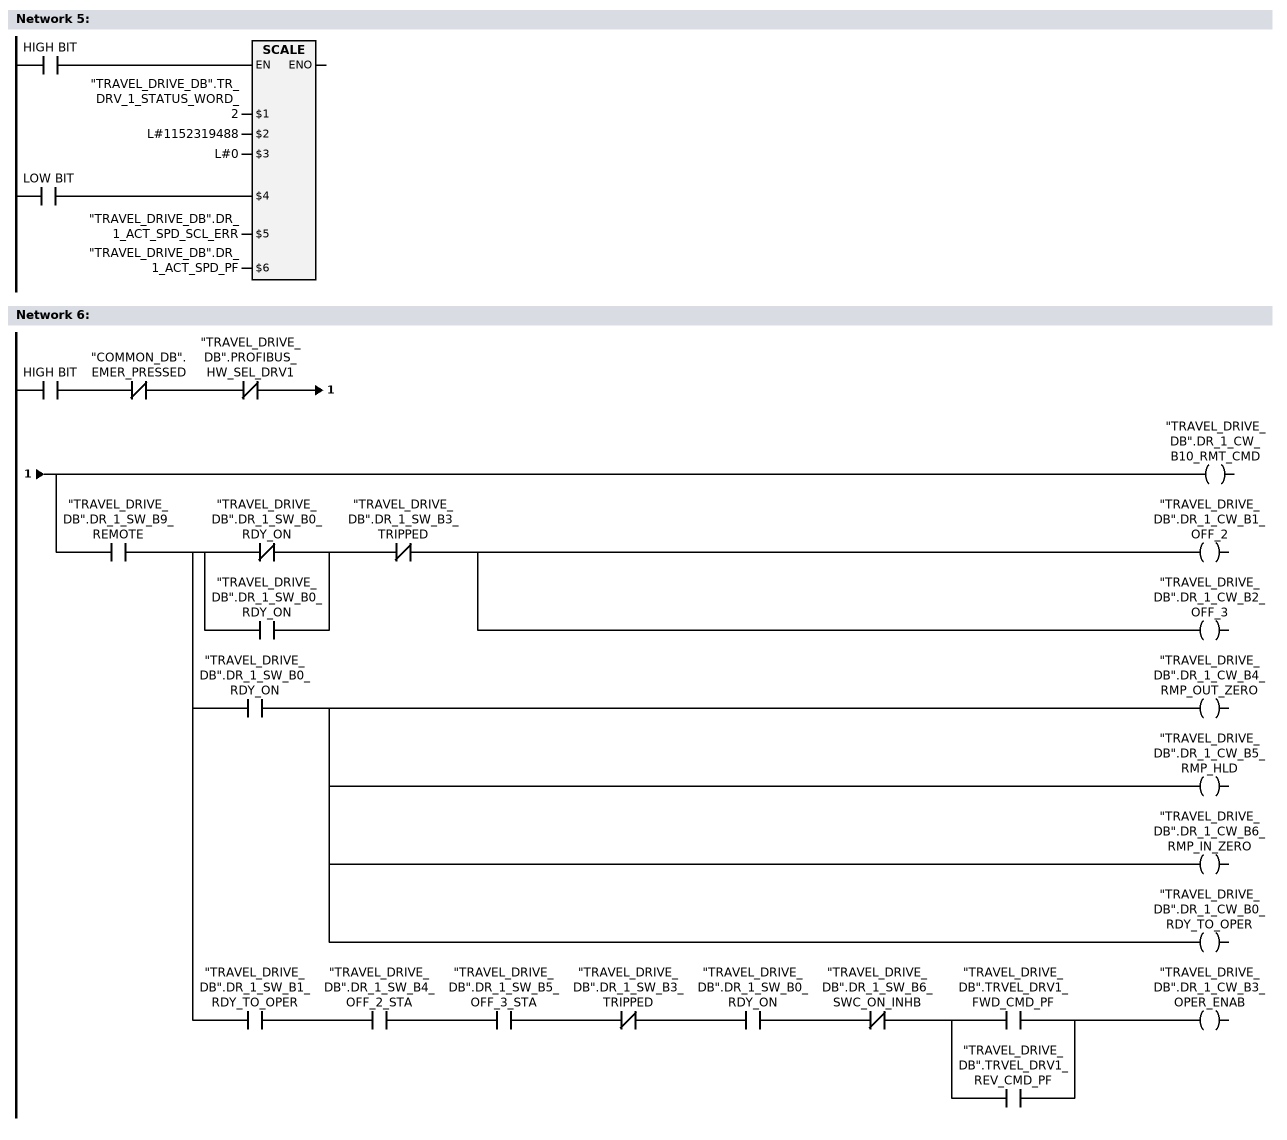
NETWORK
TITLE =
      A     "LOW BIT";
      =     L 22.0;
      BLD   103;
      A     "HIGH BIT";
      JNB   M007;
      CALL  "SCALE" (
           $1                       := "TRAVEL_DRIVE_DB".TR_DRV_1_STATUS_WORD_2,
           $2                       := L#1152319488,
           $3                       := L#0,
           $4                       := L 22.0,
           $5                       := "TRAVEL_DRIVE_DB".DR_1_ACT_SPD_SCL_ERR,
           $6                       := "TRAVEL_DRIVE_DB".DR_1_ACT_SPD_PF);
M007: NOP   0;
NETWORK
TITLE =
      A     "HIGH BIT";
      AN    "COMMON_DB".EMER_PRESSED;
      AN    "TRAVEL_DRIVE_DB".PROFIBUS_HW_SEL_DRV1;
      =     L 22.0;
      A     L 22.0;
      BLD   102;
      =     "TRAVEL_DRIVE_DB".DR_1_CW_B10_RMT_CMD;
      A     L 22.0;
      A     "TRAVEL_DRIVE_DB".DR_1_SW_B9_REMOTE;
      =     L 22.1;
      A     L 22.1;
      A(;
      ON    "TRAVEL_DRIVE_DB".DR_1_SW_B0_RDY_ON;
      O     "TRAVEL_DRIVE_DB".DR_1_SW_B0_RDY_ON;
      );
      AN    "TRAVEL_DRIVE_DB".DR_1_SW_B3_TRIPPED;
      =     "TRAVEL_DRIVE_DB".DR_1_CW_B1_OFF_2;
      =     "TRAVEL_DRIVE_DB".DR_1_CW_B2_OFF_3;
      A     L 22.1;
      A     "TRAVEL_DRIVE_DB".DR_1_SW_B0_RDY_ON;
      =     "TRAVEL_DRIVE_DB".DR_1_CW_B4_RMP_OUT_ZERO;
      =     "TRAVEL_DRIVE_DB".DR_1_CW_B5_RMP_HLD;
      =     "TRAVEL_DRIVE_DB".DR_1_CW_B6_RMP_IN_ZERO;
      =     "TRAVEL_DRIVE_DB".DR_1_CW_B0_RDY_TO_OPER;
      A     L 22.1;
      A     "TRAVEL_DRIVE_DB".DR_1_SW_B1_RDY_TO_OPER;
      A     "TRAVEL_DRIVE_DB".DR_1_SW_B4_OFF_2_STA;
      A     "TRAVEL_DRIVE_DB".DR_1_SW_B5_OFF_3_STA;
      AN    "TRAVEL_DRIVE_DB".DR_1_SW_B3_TRIPPED;
      A     "TRAVEL_DRIVE_DB".DR_1_SW_B0_RDY_ON;
      AN    "TRAVEL_DRIVE_DB".DR_1_SW_B6_SWC_ON_INHB;
      A(;
      O     "TRAVEL_DRIVE_DB".TRVEL_DRV1_FWD_CMD_PF;
      O     "TRAVEL_DRIVE_DB".TRVEL_DRV1_REV_CMD_PF;
      );
      =     "TRAVEL_DRIVE_DB".DR_1_CW_B3_OPER_ENAB;
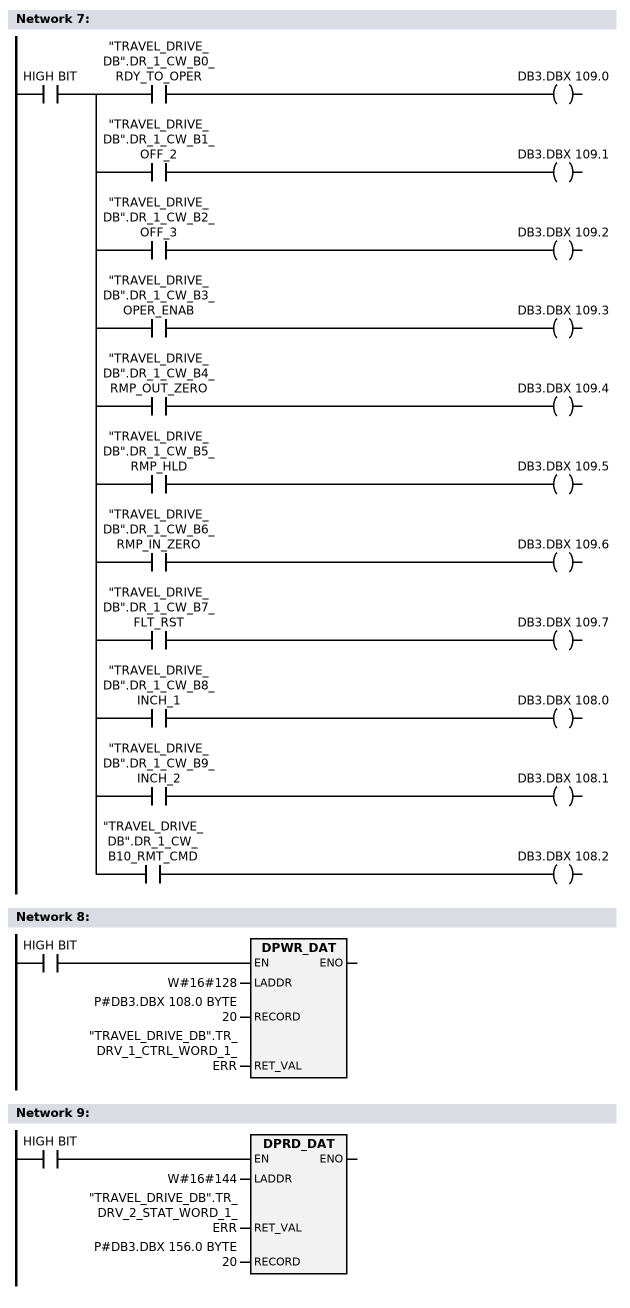
NETWORK
TITLE =
      A     "HIGH BIT";
      =     L 22.0;
      A     L 22.0;
      A     "TRAVEL_DRIVE_DB".DR_1_CW_B0_RDY_TO_OPER;
      =     DB3.DBX 109.0;
      A     L 22.0;
      A     "TRAVEL_DRIVE_DB".DR_1_CW_B1_OFF_2;
      =     DB3.DBX 109.1;
      A     L 22.0;
      A     "TRAVEL_DRIVE_DB".DR_1_CW_B2_OFF_3;
      =     DB3.DBX 109.2;
      A     L 22.0;
      A     "TRAVEL_DRIVE_DB".DR_1_CW_B3_OPER_ENAB;
      =     DB3.DBX 109.3;
      A     L 22.0;
      A     "TRAVEL_DRIVE_DB".DR_1_CW_B4_RMP_OUT_ZERO;
      =     DB3.DBX 109.4;
      A     L 22.0;
      A     "TRAVEL_DRIVE_DB".DR_1_CW_B5_RMP_HLD;
      =     DB3.DBX 109.5;
      A     L 22.0;
      A     "TRAVEL_DRIVE_DB".DR_1_CW_B6_RMP_IN_ZERO;
      =     DB3.DBX 109.6;
      A     L 22.0;
      A     "TRAVEL_DRIVE_DB".DR_1_CW_B7_FLT_RST;
      =     DB3.DBX 109.7;
      A     L 22.0;
      A     "TRAVEL_DRIVE_DB".DR_1_CW_B8_INCH_1;
      =     DB3.DBX 108.0;
      A     L 22.0;
      A     "TRAVEL_DRIVE_DB".DR_1_CW_B9_INCH_2;
      =     DB3.DBX 108.1;
      A     L 22.0;
      A     "TRAVEL_DRIVE_DB".DR_1_CW_B10_RMT_CMD;
      =     DB3.DBX 108.2;
NETWORK
TITLE =
      A     "HIGH BIT";
      JNB   M008;
      CALL  "DPWR_DAT" (
           LADDR                    := W#16#128,
           RECORD                   := P#DB3.DBX 108.0 BYTE 20,
           RET_VAL                  := "TRAVEL_DRIVE_DB".TR_DRV_1_CTRL_WORD_1_ERR);
M008: NOP   0;
NETWORK
TITLE =
      A     "HIGH BIT";
      JNB   M009;
      CALL  "DPRD_DAT" (
           LADDR                    := W#16#144,
           RET_VAL                  := "TRAVEL_DRIVE_DB".TR_DRV_2_STAT_WORD_1_ERR,
           RECORD                   := P#DB3.DBX 156.0 BYTE 20);
M009: NOP   0;
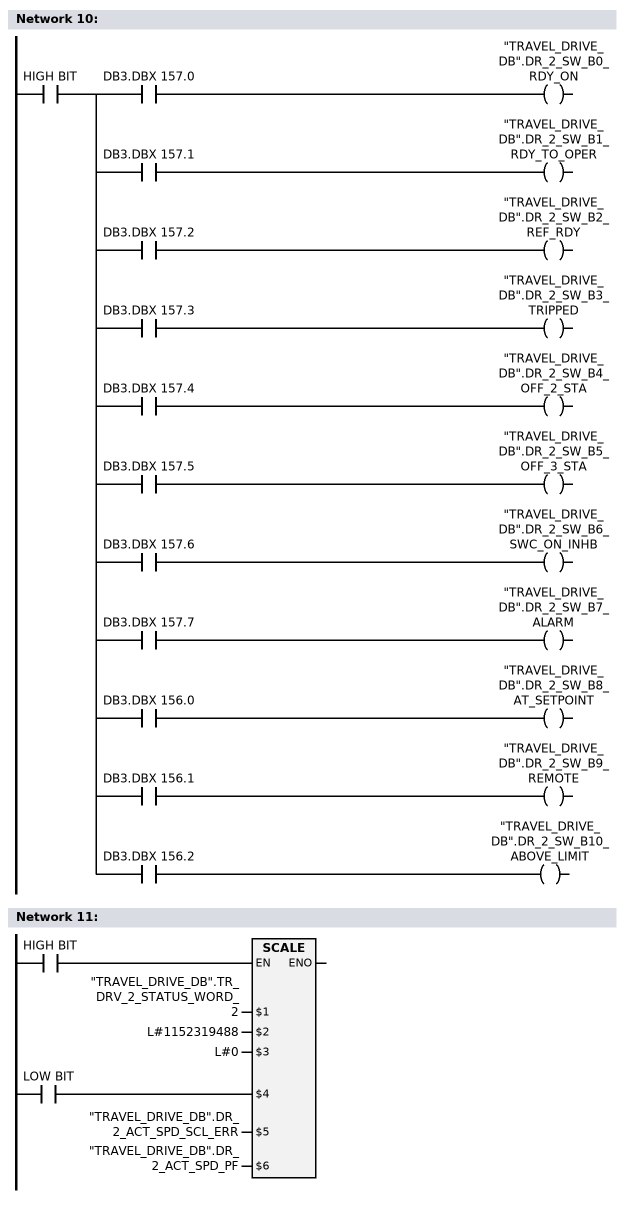
NETWORK
TITLE =
      A     "HIGH BIT";
      =     L 22.0;
      A     L 22.0;
      A     DB3.DBX 157.0;
      =     "TRAVEL_DRIVE_DB".DR_2_SW_B0_RDY_ON;
      A     L 22.0;
      A     DB3.DBX 157.1;
      =     "TRAVEL_DRIVE_DB".DR_2_SW_B1_RDY_TO_OPER;
      A     L 22.0;
      A     DB3.DBX 157.2;
      =     "TRAVEL_DRIVE_DB".DR_2_SW_B2_REF_RDY;
      A     L 22.0;
      A     DB3.DBX 157.3;
      =     "TRAVEL_DRIVE_DB".DR_2_SW_B3_TRIPPED;
      A     L 22.0;
      A     DB3.DBX 157.4;
      =     "TRAVEL_DRIVE_DB".DR_2_SW_B4_OFF_2_STA;
      A     L 22.0;
      A     DB3.DBX 157.5;
      =     "TRAVEL_DRIVE_DB".DR_2_SW_B5_OFF_3_STA;
      A     L 22.0;
      A     DB3.DBX 157.6;
      =     "TRAVEL_DRIVE_DB".DR_2_SW_B6_SWC_ON_INHB;
      A     L 22.0;
      A     DB3.DBX 157.7;
      =     "TRAVEL_DRIVE_DB".DR_2_SW_B7_ALARM;
      A     L 22.0;
      A     DB3.DBX 156.0;
      =     "TRAVEL_DRIVE_DB".DR_2_SW_B8_AT_SETPOINT;
      A     L 22.0;
      A     DB3.DBX 156.1;
      =     "TRAVEL_DRIVE_DB".DR_2_SW_B9_REMOTE;
      A     L 22.0;
      A     DB3.DBX 156.2;
      =     "TRAVEL_DRIVE_DB".DR_2_SW_B10_ABOVE_LIMIT;
NETWORK
TITLE =
      A     "LOW BIT";
      =     L 22.0;
      BLD   103;
      A     "HIGH BIT";
      JNB   M010;
      CALL  "SCALE" (
           $1                       := "TRAVEL_DRIVE_DB".TR_DRV_2_STATUS_WORD_2,
           $2                       := L#1152319488,
           $3                       := L#0,
           $4                       := L 22.0,
           $5                       := "TRAVEL_DRIVE_DB".DR_2_ACT_SPD_SCL_ERR,
           $6                       := "TRAVEL_DRIVE_DB".DR_2_ACT_SPD_PF);
M010: NOP   0;
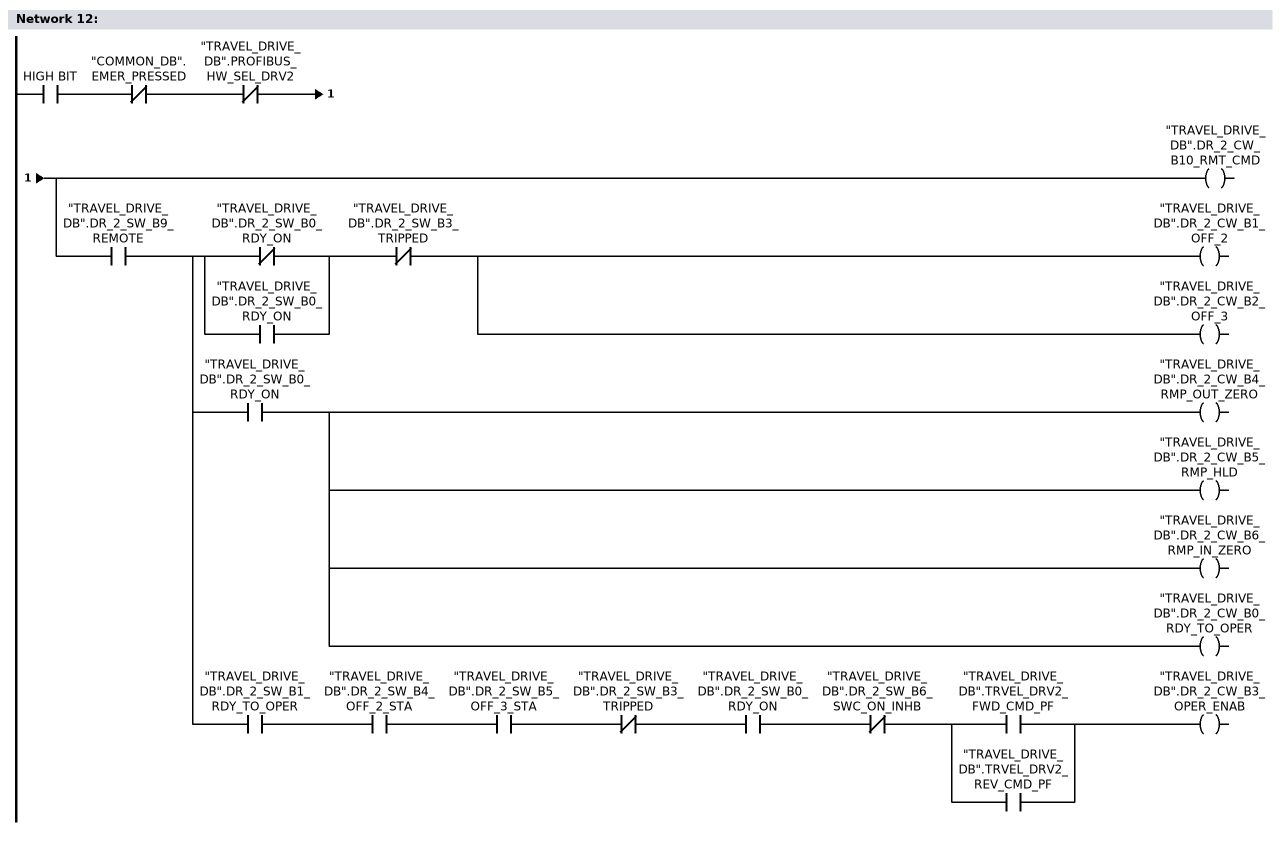
NETWORK
TITLE =
      A     "HIGH BIT";
      AN    "COMMON_DB".EMER_PRESSED;
      AN    "TRAVEL_DRIVE_DB".PROFIBUS_HW_SEL_DRV2;
      =     L 22.0;
      A     L 22.0;
      BLD   102;
      =     "TRAVEL_DRIVE_DB".DR_2_CW_B10_RMT_CMD;
      A     L 22.0;
      A     "TRAVEL_DRIVE_DB".DR_2_SW_B9_REMOTE;
      =     L 22.1;
      A     L 22.1;
      A(;
      ON    "TRAVEL_DRIVE_DB".DR_2_SW_B0_RDY_ON;
      O     "TRAVEL_DRIVE_DB".DR_2_SW_B0_RDY_ON;
      );
      AN    "TRAVEL_DRIVE_DB".DR_2_SW_B3_TRIPPED;
      =     "TRAVEL_DRIVE_DB".DR_2_CW_B1_OFF_2;
      =     "TRAVEL_DRIVE_DB".DR_2_CW_B2_OFF_3;
      A     L 22.1;
      A     "TRAVEL_DRIVE_DB".DR_2_SW_B0_RDY_ON;
      =     "TRAVEL_DRIVE_DB".DR_2_CW_B4_RMP_OUT_ZERO;
      =     "TRAVEL_DRIVE_DB".DR_2_CW_B5_RMP_HLD;
      =     "TRAVEL_DRIVE_DB".DR_2_CW_B6_RMP_IN_ZERO;
      =     "TRAVEL_DRIVE_DB".DR_2_CW_B0_RDY_TO_OPER;
      A     L 22.1;
      A     "TRAVEL_DRIVE_DB".DR_2_SW_B1_RDY_TO_OPER;
      A     "TRAVEL_DRIVE_DB".DR_2_SW_B4_OFF_2_STA;
      A     "TRAVEL_DRIVE_DB".DR_2_SW_B5_OFF_3_STA;
      AN    "TRAVEL_DRIVE_DB".DR_2_SW_B3_TRIPPED;
      A     "TRAVEL_DRIVE_DB".DR_2_SW_B0_RDY_ON;
      AN    "TRAVEL_DRIVE_DB".DR_2_SW_B6_SWC_ON_INHB;
      A(;
      O     "TRAVEL_DRIVE_DB".TRVEL_DRV2_FWD_CMD_PF;
      O     "TRAVEL_DRIVE_DB".TRVEL_DRV2_REV_CMD_PF;
      );
      =     "TRAVEL_DRIVE_DB".DR_2_CW_B3_OPER_ENAB;
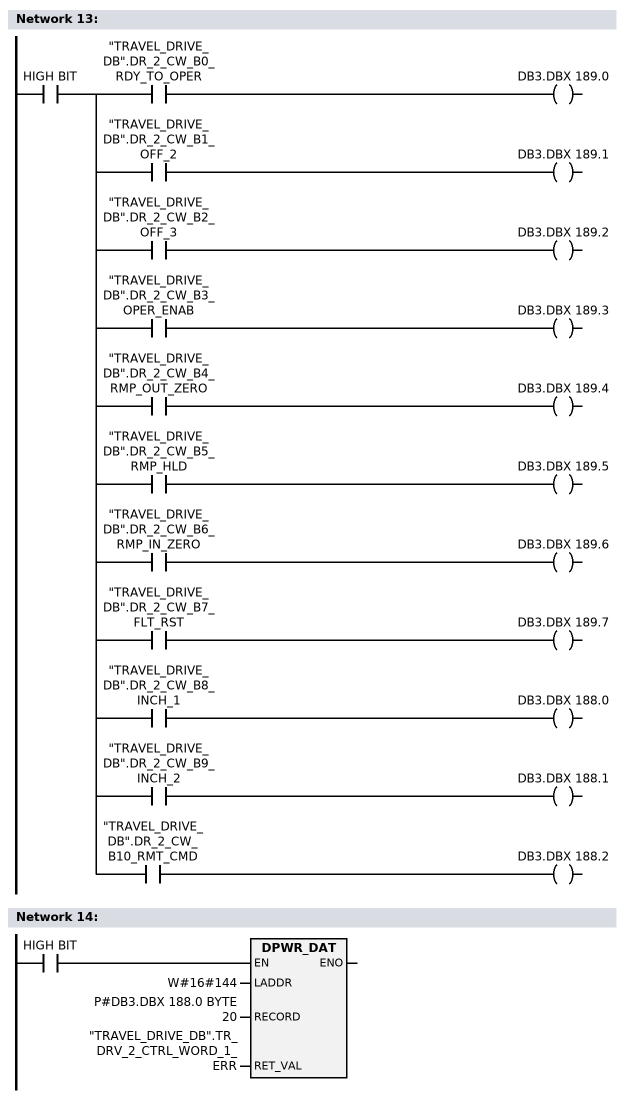
NETWORK
TITLE =
      A     "HIGH BIT";
      =     L 22.0;
      A     L 22.0;
      A     "TRAVEL_DRIVE_DB".DR_2_CW_B0_RDY_TO_OPER;
      =     DB3.DBX 189.0;
      A     L 22.0;
      A     "TRAVEL_DRIVE_DB".DR_2_CW_B1_OFF_2;
      =     DB3.DBX 189.1;
      A     L 22.0;
      A     "TRAVEL_DRIVE_DB".DR_2_CW_B2_OFF_3;
      =     DB3.DBX 189.2;
      A     L 22.0;
      A     "TRAVEL_DRIVE_DB".DR_2_CW_B3_OPER_ENAB;
      =     DB3.DBX 189.3;
      A     L 22.0;
      A     "TRAVEL_DRIVE_DB".DR_2_CW_B4_RMP_OUT_ZERO;
      =     DB3.DBX 189.4;
      A     L 22.0;
      A     "TRAVEL_DRIVE_DB".DR_2_CW_B5_RMP_HLD;
      =     DB3.DBX 189.5;
      A     L 22.0;
      A     "TRAVEL_DRIVE_DB".DR_2_CW_B6_RMP_IN_ZERO;
      =     DB3.DBX 189.6;
      A     L 22.0;
      A     "TRAVEL_DRIVE_DB".DR_2_CW_B7_FLT_RST;
      =     DB3.DBX 189.7;
      A     L 22.0;
      A     "TRAVEL_DRIVE_DB".DR_2_CW_B8_INCH_1;
      =     DB3.DBX 188.0;
      A     L 22.0;
      A     "TRAVEL_DRIVE_DB".DR_2_CW_B9_INCH_2;
      =     DB3.DBX 188.1;
      A     L 22.0;
      A     "TRAVEL_DRIVE_DB".DR_2_CW_B10_RMT_CMD;
      =     DB3.DBX 188.2;
NETWORK
TITLE =
      A     "HIGH BIT";
      JNB   M011;
      CALL  "DPWR_DAT" (
           LADDR                    := W#16#144,
           RECORD                   := P#DB3.DBX 188.0 BYTE 20,
           RET_VAL                  := "TRAVEL_DRIVE_DB".TR_DRV_2_CTRL_WORD_1_ERR);
M011: NOP   0;
END_FUNCTION

FUNCTION "TATA_COMMUNICATION" : VOID	// FC 11
AUTHOR : Kamillas
VERSION : 0.1
BEGIN
// (block stored without names or comments; labels and parameter names are numbered)
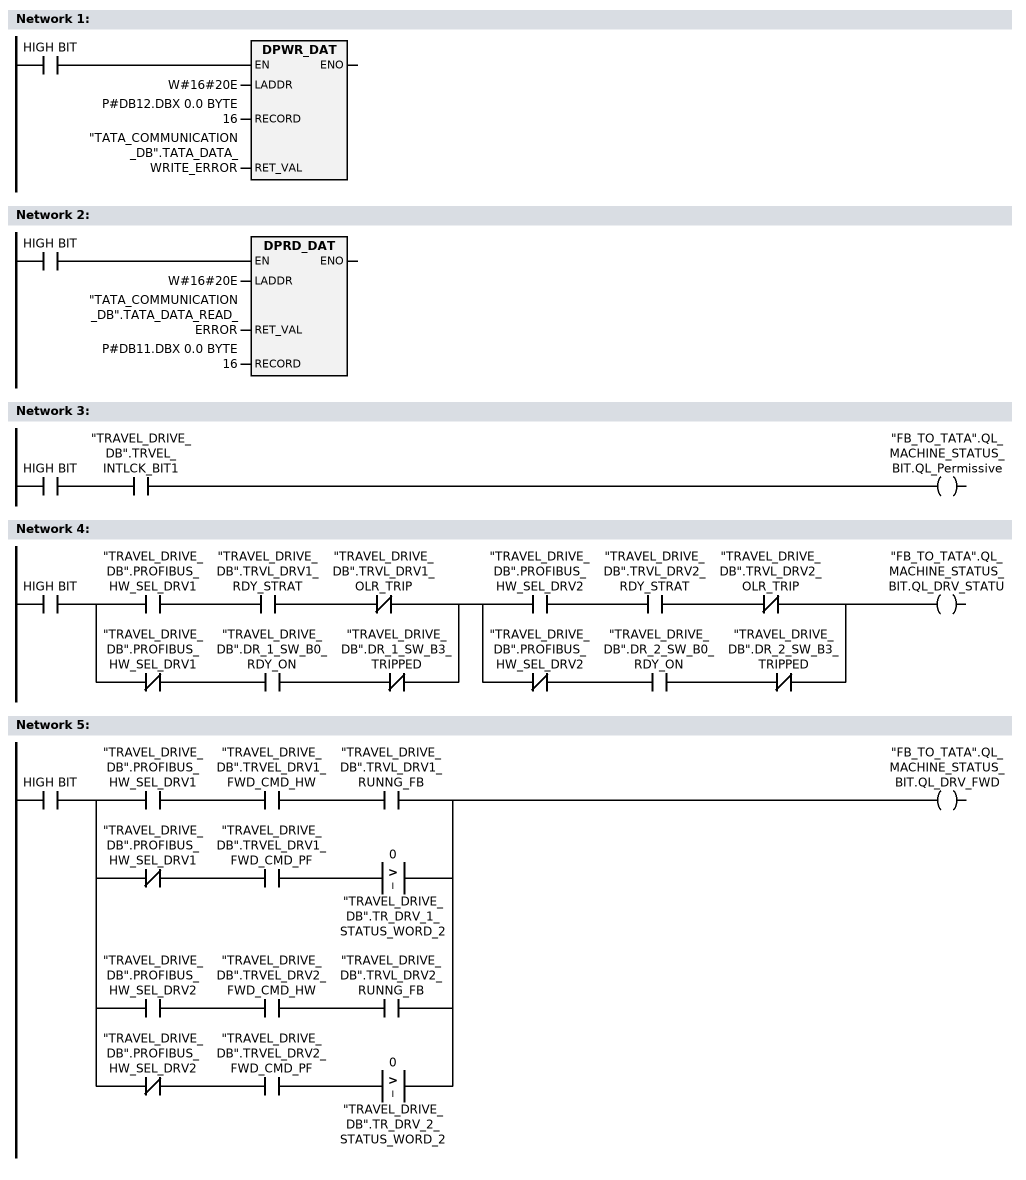
NETWORK
TITLE =
      A     "HIGH BIT";
      JNB   M001;
      CALL  "DPWR_DAT" (
           LADDR                    := W#16#20E,
           RECORD                   := P#DB12.DBX 0.0 BYTE 16,
           RET_VAL                  := "TATA_COMMUNICATION_DB".TATA_DATA_WRITE_ERROR);
M001: NOP   0;
NETWORK
TITLE =
      A     "HIGH BIT";
      JNB   M002;
      CALL  "DPRD_DAT" (
           LADDR                    := W#16#20E,
           RET_VAL                  := "TATA_COMMUNICATION_DB".TATA_DATA_READ_ERROR,
           RECORD                   := P#DB11.DBX 0.0 BYTE 16);
M002: NOP   0;
NETWORK
TITLE =
      A     "HIGH BIT";
      A     "TRAVEL_DRIVE_DB".TRVEL_INTLCK_BIT1;
      =     "FB_TO_TATA".QL_MACHINE_STATUS_BIT.QL_Permissive;
NETWORK
TITLE =
      A     "HIGH BIT";
      A(;
      A     "TRAVEL_DRIVE_DB".PROFIBUS_HW_SEL_DRV1;
      A     "TRAVEL_DRIVE_DB".TRVL_DRV1_RDY_STRAT;
      AN    "TRAVEL_DRIVE_DB".TRVL_DRV1_OLR_TRIP;
      O;
      AN    "TRAVEL_DRIVE_DB".PROFIBUS_HW_SEL_DRV1;
      A     "TRAVEL_DRIVE_DB".DR_1_SW_B0_RDY_ON;
      AN    "TRAVEL_DRIVE_DB".DR_1_SW_B3_TRIPPED;
      );
      A(;
      A     "TRAVEL_DRIVE_DB".PROFIBUS_HW_SEL_DRV2;
      A     "TRAVEL_DRIVE_DB".TRVL_DRV2_RDY_STRAT;
      AN    "TRAVEL_DRIVE_DB".TRVL_DRV2_OLR_TRIP;
      O;
      AN    "TRAVEL_DRIVE_DB".PROFIBUS_HW_SEL_DRV2;
      A     "TRAVEL_DRIVE_DB".DR_2_SW_B0_RDY_ON;
      AN    "TRAVEL_DRIVE_DB".DR_2_SW_B3_TRIPPED;
      );
      =     "FB_TO_TATA".QL_MACHINE_STATUS_BIT.QL_DRV_STATU;
NETWORK
TITLE =
      A     "HIGH BIT";
      A(;
      A     "TRAVEL_DRIVE_DB".PROFIBUS_HW_SEL_DRV1;
      A     "TRAVEL_DRIVE_DB".TRVEL_DRV1_FWD_CMD_HW;
      A     "TRAVEL_DRIVE_DB".TRVL_DRV1_RUNNG_FB;
      O;
      AN    "TRAVEL_DRIVE_DB".PROFIBUS_HW_SEL_DRV1;
      A     "TRAVEL_DRIVE_DB".TRVEL_DRV1_FWD_CMD_PF;
      A(;
      L     0;
      L     "TRAVEL_DRIVE_DB".TR_DRV_1_STATUS_WORD_2;
      >I;
      );
      O;
      A     "TRAVEL_DRIVE_DB".PROFIBUS_HW_SEL_DRV2;
      A     "TRAVEL_DRIVE_DB".TRVEL_DRV2_FWD_CMD_HW;
      A     "TRAVEL_DRIVE_DB".TRVL_DRV2_RUNNG_FB;
      O;
      AN    "TRAVEL_DRIVE_DB".PROFIBUS_HW_SEL_DRV2;
      A     "TRAVEL_DRIVE_DB".TRVEL_DRV2_FWD_CMD_PF;
      A(;
      L     0;
      L     "TRAVEL_DRIVE_DB".TR_DRV_2_STATUS_WORD_2;
      >I;
      );
      );
      =     "FB_TO_TATA".QL_MACHINE_STATUS_BIT.QL_DRV_FWD;
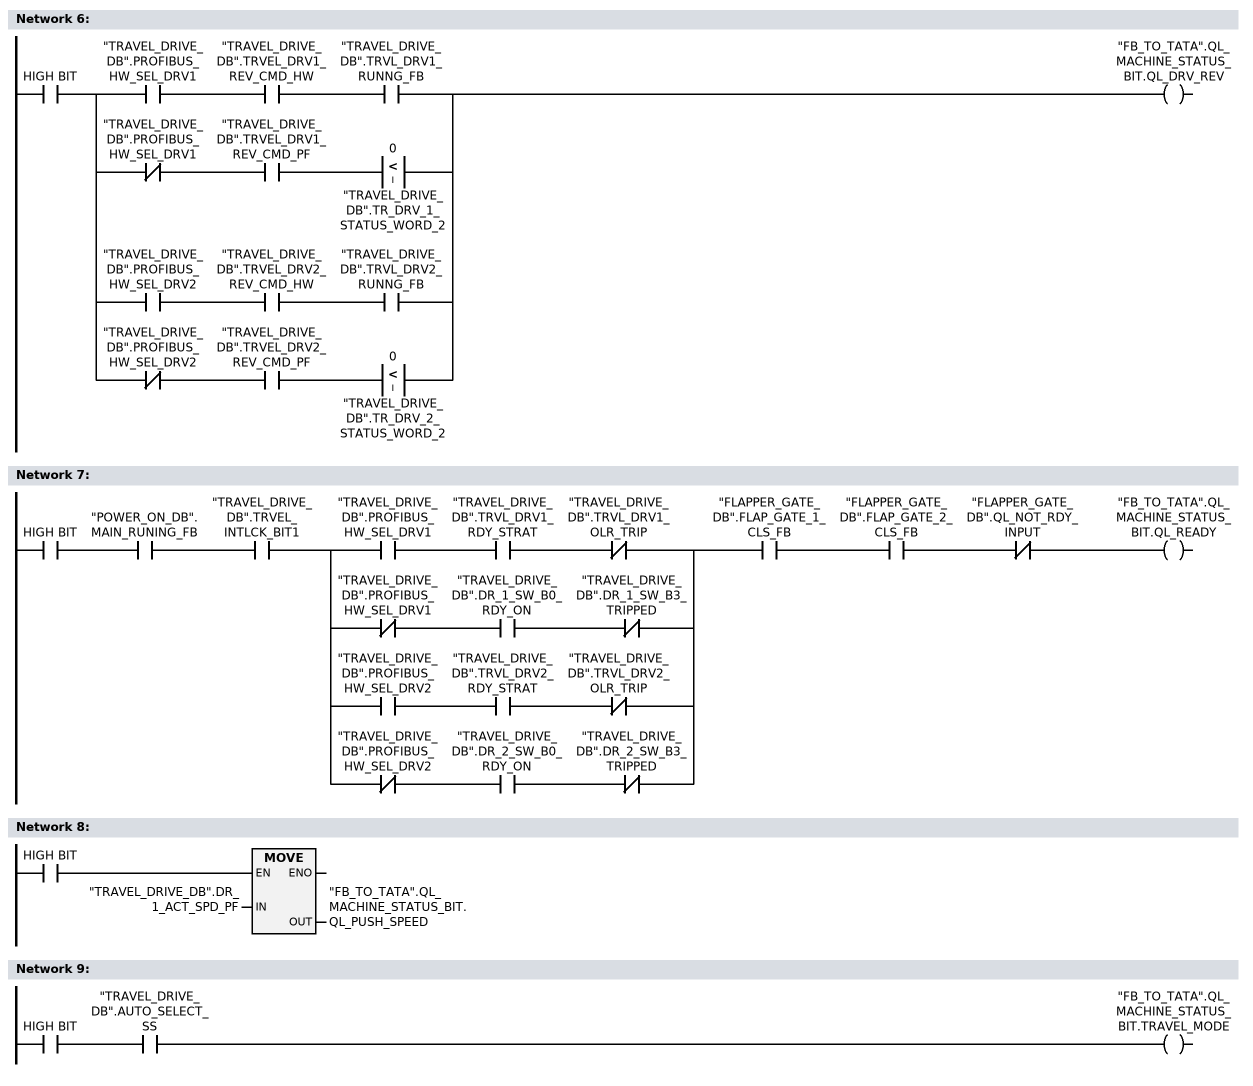
NETWORK
TITLE =
      A     "HIGH BIT";
      A(;
      A     "TRAVEL_DRIVE_DB".PROFIBUS_HW_SEL_DRV1;
      A     "TRAVEL_DRIVE_DB".TRVEL_DRV1_REV_CMD_HW;
      A     "TRAVEL_DRIVE_DB".TRVL_DRV1_RUNNG_FB;
      O;
      AN    "TRAVEL_DRIVE_DB".PROFIBUS_HW_SEL_DRV1;
      A     "TRAVEL_DRIVE_DB".TRVEL_DRV1_REV_CMD_PF;
      A(;
      L     0;
      L     "TRAVEL_DRIVE_DB".TR_DRV_1_STATUS_WORD_2;
      <I;
      );
      O;
      A     "TRAVEL_DRIVE_DB".PROFIBUS_HW_SEL_DRV2;
      A     "TRAVEL_DRIVE_DB".TRVEL_DRV2_REV_CMD_HW;
      A     "TRAVEL_DRIVE_DB".TRVL_DRV2_RUNNG_FB;
      O;
      AN    "TRAVEL_DRIVE_DB".PROFIBUS_HW_SEL_DRV2;
      A     "TRAVEL_DRIVE_DB".TRVEL_DRV2_REV_CMD_PF;
      A(;
      L     0;
      L     "TRAVEL_DRIVE_DB".TR_DRV_2_STATUS_WORD_2;
      <I;
      );
      );
      =     "FB_TO_TATA".QL_MACHINE_STATUS_BIT.QL_DRV_REV;
NETWORK
TITLE =
      A     "HIGH BIT";
      A     "POWER_ON_DB".MAIN_RUNING_FB;
      A     "TRAVEL_DRIVE_DB".TRVEL_INTLCK_BIT1;
      A(;
      A     "TRAVEL_DRIVE_DB".PROFIBUS_HW_SEL_DRV1;
      A     "TRAVEL_DRIVE_DB".TRVL_DRV1_RDY_STRAT;
      AN    "TRAVEL_DRIVE_DB".TRVL_DRV1_OLR_TRIP;
      O;
      AN    "TRAVEL_DRIVE_DB".PROFIBUS_HW_SEL_DRV1;
      A     "TRAVEL_DRIVE_DB".DR_1_SW_B0_RDY_ON;
      AN    "TRAVEL_DRIVE_DB".DR_1_SW_B3_TRIPPED;
      O;
      A     "TRAVEL_DRIVE_DB".PROFIBUS_HW_SEL_DRV2;
      A     "TRAVEL_DRIVE_DB".TRVL_DRV2_RDY_STRAT;
      AN    "TRAVEL_DRIVE_DB".TRVL_DRV2_OLR_TRIP;
      O;
      AN    "TRAVEL_DRIVE_DB".PROFIBUS_HW_SEL_DRV2;
      A     "TRAVEL_DRIVE_DB".DR_2_SW_B0_RDY_ON;
      AN    "TRAVEL_DRIVE_DB".DR_2_SW_B3_TRIPPED;
      );
      A     "FLAPPER_GATE_DB".FLAP_GATE_1_CLS_FB;
      A     "FLAPPER_GATE_DB".FLAP_GATE_2_CLS_FB;
      AN    "FLAPPER_GATE_DB".QL_NOT_RDY_INPUT;
      =     "FB_TO_TATA".QL_MACHINE_STATUS_BIT.QL_READY;
NETWORK
TITLE =
      A     "HIGH BIT";
      JNB   M003;
      L     "TRAVEL_DRIVE_DB".DR_1_ACT_SPD_PF;
      T     "FB_TO_TATA".QL_MACHINE_STATUS_BIT.QL_PUSH_SPEED;
M003: NOP   0;
NETWORK
TITLE =
      A     "HIGH BIT";
      A     "TRAVEL_DRIVE_DB".AUTO_SELECT_SS;
      =     "FB_TO_TATA".QL_MACHINE_STATUS_BIT.TRAVEL_MODE;
END_FUNCTION

// FC 105: know-how protected block, not included

// FC 106: know-how protected block, not included

DATA_BLOCK "REV_END_POSITION"	// DB 1
VERSION : 0.1
  STRUCT
   MAIN_RUN_FB : BOOL ;	//MAIN POWER RUNNING FEED BACK
   CONTROL_ON_FB : BOOL ;	//CONTROL POWER O FEED BACK
   EMERGENCY_PB_AT_CD : BOOL ;	//EMERGENCY STOP PUSHBUTTON AT CD
   LAMP_TEST_PB_AT_CD : BOOL ;	//LAMP TEST PUSHBUTTON AT CD
   ALARM_ACT_PB_CD : BOOL ;	//ALARM ACKNOLODGE PUSH BUTTON AT CD
   MANUAL_SELECT_SS : BOOL ;	//MANUAL MODE SELECTION
   AUTO_SS : BOOL ;	//AUTO MODE SELECTION
   CRIP_SPD_SS : BOOL ;	//CRIPPING SPEED SELECTOR SPEED
   PROFIBUS_HW_SEL_DRV1 : BOOL ;	//PROFIBUS/HARDWARE SELECTION DRIVE1
   TRVL_DRV1_RDY : BOOL ;	//TRAVEL DRIVE 1 READY TO START
   TRVL_DRV1_RUN_FB : BOOL ;	//TRAVEL DRIVE 1 RUNNING FEED BACK
   TRVL_DRV1_OLR_TRIP : BOOL ;	//TRAVEL DRIVE 1 TRIP FEED BACK
   PROFIBUS_HW_SEL_DRV2 : BOOL ;	//PROFIBUS/HARDWARE SELECTION DRIVE2
   TRVL_DRV2_RDY : BOOL ;	//TRAVEL DRIVE 2 READY TO START
   TRVL_DRV2_RUN_FB : BOOL ;	//TRAVEL DRIVE 2 RUNNING FEED BACK
   TRVL_DRV2_OLR_TRIP : BOOL ;	//TRAVEL DRIVE 2 TRIP FEED BACK
   CREPING_SPEED_FB : BOOL ;	//CREEPING SPEED FEED BACK
   K_ZERO_PWR_OFF : BOOL ;	//ZERO SPEED IN LONG TRAVEL MODE LIMIT SWITCH
   JOY_ST_DEADMAN_BUTTON : BOOL ;	//JOYSTICK DEADMAN BUTTON
   JOY_ST_HOME_POSITN : BOOL ;	//JOYSTICK HOME POSITION
   JOY_ST_FWD_POSITN : BOOL ;	//JOYSTICK FORWARD POSITION
   JOY_ST_REV_POSITN : BOOL ;	//JOYSTICK REVERSE POSITION
   EMERGENCY_PB_AT_MCC : BOOL ;	//EMERGENCY STOP PUSHBUTTON AT MCC
   SPARE_4 : BOOL ;	//SPARE 4
   FWD_END_LIMIT_SW_FB : BOOL ;	//FORWARD END LIMIT SWITCH FEED BACK
   FWD_EMER_END_LIMIT_SW_FB : BOOL ;	//FORWARD EMERGENCY END LIMIT SWITCH FEED BACK
   REV_END_LIMIT_SW_FB : BOOL ;	//REVERSE END LIMIT SWITCH FEED BACK
   REV_EMER_END_LIMIT_SW_FB : BOOL ;	//REVERSE EMERGENCY END LIMIT SWITCH FEED BACK
   FLAP_GATE_1_CLS : BOOL ;	//FLAPPER GATE 1 CLOSE FEEDBACK
   FLAP_GATE_2_CLS : BOOL ;	//FLAPPER GATE 2 CLOSE FEEDBACK
   SPARE_INPUT1 : BOOL ;	//SPARE INPUT 1
   SPARE_INPUT2 : BOOL ;	//SPARE INPUT 2
   COMPRSR_1_RDY_START : BOOL ;	//COMPRESSOR 1 READY TO START
   COMPRSR_1_RUNG_FB : BOOL ;	//COMPRESSOR 1 RUNNING FEED BACK
   COMPRSR_2_RDY_START : BOOL ;	//COMPRESSOR 2 READY TO START
   COMPRSR_2_RUNG_FB : BOOL ;	//COMPRESSOR 2 RUNNING FEED BACK
   COMPRSR_1_2_SEL_SW : BOOL ;	//COMPRESSOR 1 & 2 SELECTION
   COMPRSR_1_START_PB : BOOL ;	//COMPRESSOR 1 START PUSH BUTTON
   COMPRSR_1_STOP_PB : BOOL ;	//COMPRESSOR 1 STOP PUSH BUTTON
   CD_PC_SEL : BOOL ;	//CD OR PC SELECTION
   COMPRSR_2_START_PB : BOOL ;	//COMPRESSOR 2 START PUSH BUTTON
   COMPRSR_2_STOP_PB : BOOL ;	//COMPRESSOR 2 STOP PUSH BUTTON
   COMPRSR_MAX_PR_SW_FB : BOOL ;	//COMPRESSOR MAXIMUM PRESSURE SWITCH FEED BACK
   COMPRSR_MIN_PR_SW_FB : BOOL ;	//COMPRESSOR MINIMUM PRESSURE SWITCH FEED BACK
   COMPRSR_BRK_PR_SW_FB : BOOL ;	//COMPRESSOR BREAK LINE PRESSURE SWITCH FEED BACK
   COMPRSR_CONTROL_PR_SW_FB : BOOL ;	//COMPRESSOR CONTROL PRESSURE SWITCH FEED BACK
   SPARE_INPUT_5_6 : BOOL ;	//SPARE INPUT I5.6
   SPARE_INPUT_5_7 : BOOL ;	//SPARE INPUT I5.7
   SPARE_INPUT_6_0 : BOOL ;	//SPARE INPUT I6.0
   SIG_START_INPUT : BOOL ;	//SIGNALLING START PUSH BUTTON
   SPARE_INPUT_6_2 : BOOL ;	//SPARE INPUT I6.2
   SPARE_INPUT_6_3 : BOOL ;	//SPARE INPUT I6.3
   SPARE_INPUT_6_4 : BOOL ;	//SPARE INPUT I6.4
   SPARE_INPUT_6_5 : BOOL ;	//SPARE INPUT I6.5
   SPARE_INPUT_6_6 : BOOL ;	//SPARE INPUT I6.6
   SPARE_INPUT_6_7 : BOOL ;	//SPARE INPUT I6.7
   SPARE_INPUT_7_0 : BOOL ;	//SPARE INPUT I7.0
   SPARE_INPUT_7_1 : BOOL ;	//SPARE INPUT I7.1
   SPARE_INPUT_7_2 : BOOL ;	//SPARE INPUT I7.2
   SPARE_INPUT_7_3 : BOOL ;	//SPARE INPUT I7.3
   SPARE_INPUT_7_4 : BOOL ;	//SPARE INPUT I7.4
   SPARE_INPUT_7_5 : BOOL ;	//SPARE INPUT I7.5
   SPARE_INPUT_7_6 : BOOL ;	//SPARE INPUT I7.6
   SPARE_INPUT_7_7 : BOOL ;	//SPARE INPUT I7.7
  END_STRUCT ;	
BEGIN
END_DATA_BLOCK

DATA_BLOCK "OUTPUT_MAPPING_DB"	// DB 2
VERSION : 0.1
  STRUCT
   MAIN_PWR_START_CMD : BOOL ;	//MAIN POWER START COMMEND
   CONTROL_ON_IND : BOOL ;	//CONTROL POWER ON INDICATION
   AUTO_POSITION_ACK_IND : BOOL ;	//AUTO POSITION ACKNOWLEDGEMENT INDICATION
   TRVL_DRV_1_FWD_CMD1 : BOOL ;	//TRAVEL DRIVE 1 FORWARD COMMEND
   TRVL_DRV_1_REV_CMD1 : BOOL ;	//TRAVEL DRIVE 1 REVERSE COMMEND
   TRVL_DRV_2_FWD_CMD1 : BOOL ;	//TRAVEL DRIVE 2 FORWARD COMMEND
   TRVL_DRV_2_REV_CMD1 : BOOL ;	//TRAVEL DRIVE 2 REVERSE COMMEND
   SPARE_OUTPUT_0_7 : BOOL ;	//SPARE OUTPUT Q0.7
   SPARE_OUTPUT_1_0 : BOOL ;	//SPARE OUTPUT Q1.0
   SPARE_OUTPUT_1_1 : BOOL ;	//SPARE OUTPUT Q1.1
   SPARE_OUTPUT_1_2 : BOOL ;	//SPARE OUTPUT Q1.2
   SPARE_OUTPUT_1_3 : BOOL ;	//SPARE OUTPUT Q1.3
   TRVL_PERMSN_IND : BOOL ;	//TRAVEL PERMISSION INDICATION
   SPARE_OUTPUT_1_5 : BOOL ;	//SPARE OUTPUT Q1.5
   SPARE_OUTPUT_1_6 : BOOL ;	//SPARE OUTPUT Q1.6
   SPARE_OUTPUT_1_7 : BOOL ;	//SPARE OUTPUT Q1.7
   CMPRSR_1_ON_CMD : BOOL ;	//COMPRESSOR 1 ON COMMEND
   CMPRSR_2_ON_CMD : BOOL ;	//COMPRESSOR 2 ON COMMEND
   CMPRSR_1_ON_IND : BOOL ;	//COMPRESSOR 1 ON INDICATION
   CMPRSR_2_ON_IND : BOOL ;	//COMPRESSOR 2 ON INDICATION
   QUEN_DEL_TIME : BOOL ;	//QUENCHING DELAY TIME Q2.4
   SPARE_OUTPUT_2_5 : BOOL ;	//SPARE OUTPUT Q2.5
   SPARE_OUTPUT_2_6 : BOOL ;	//QL_1_MIN_HIGH-BIT_FOR_PERMISSION
   SPARE_OUTPUT_2_7 : BOOL ;	//SPARE OUTPUT Q2.7
   SPARE_OUTPUT_3_0 : BOOL ;	//SPARE OUTPUT Q3.0
   SPARE_OUTPUT_3_1 : BOOL ;	//SPARE OUTPUT Q3.1
   SPARE_OUTPUT_3_2 : BOOL ;	//SPARE OUTPUT Q3.2
   SPARE_OUTPUT_3_3 : BOOL ;	//SPARE OUTPUT Q3.3
   SPARE_OUTPUT_3_4 : BOOL ;	//SPARE OUTPUT Q3.4
   SPARE_OUTPUT_3_5 : BOOL ;	//SPARE OUTPUT Q3.5
   SPARE_OUTPUT_3_6 : BOOL ;	//SPARE OUTPUT Q3.6
   SPARE_OUTPUT_3_7 : BOOL ;	//SPARE OUTPUT Q3.7
   HOOTER_ON_CMD : BOOL ;	//HOOTER ON COMMAND Q4.0
  END_STRUCT ;	
BEGIN
END_DATA_BLOCK

DATA_BLOCK "TRAVEL_DRIVE_DB"	// DB 3
VERSION : 0.1
  STRUCT
   TRVEL_DRV1_FWD_CMD : BOOL ;	//TRAVEL DRIVE1 FORWARD COMMEND
   TRVEL_DRV1_REV_CMD : BOOL ;	//TRAVEL DRIVE1 REVERSE COMMEND
   TRVEL_INTLCK_BIT : BOOL ;	//TRAVEL DRIVE INTERLOCK BIT
   TRVEL_DRV2_FWD_CMD : BOOL ;	//TRAVEL DRIVE2 FORWARD COMMEND
   TRVEL_DRV2_REV_CMD : BOOL ;	//TRAVEL DRIVE2 REVERSE COMMEND
   TRVEL_INTLCK_BIT1 : BOOL ;	//TRAVEL DRIVE INTERLOCK BIT1
   TRVEL_DRV1_ON_CMD : BOOL ;	//TRAVEL DRIVE1 ON COMMEND
   TRVEL_DRV2_ON_CMD : BOOL ;	//TRAVEL DRIVE2 ON COMMEND
   QUNCHING_TIME_OFF_BIT : BOOL ;	//QUNCHING TIMER OFF BIT
   QUNCHING_TIME_PLS_BIT : BOOL ;	//QUNCHING TIMER PLUSE BIT
   QUNCHING_TIME_SLOW_SPEED : BOOL ;	//QUNCHING TIMER SLOW SPEED BIT
   TRVEL_DRV1_FWD_CMD_HW : BOOL ;	//TRAVEL DRIVE1 FORWARD COMMEND HARD WARE
   TRVEL_DRV1_REV_CMD_HW : BOOL ;	//TRAVEL DRIVE1 REVERSE COMMEND HARD WARE
   TRVEL_DRV2_FWD_CMD_HW : BOOL ;	//TRAVEL DRIVE12 FORWARD COMMEND HARD WARE
   TRVEL_DRV2_REV_CMD_HW : BOOL ;	//TRAVEL DRIVE2 REVERSE COMMEND HARD WARE
   LOGO_MAX_OPERATOR_SPEED : BOOL ;	//LOCO MAXIMUM OPERATOR SPEED
   LOCO_MAX_SPEED_PROFIBUS : BOOL ;	//LOCO MAXIMUM OPERATOR SPEED IN PROFIBUS
   TRVEL_DRV1_HEALTHY_CMD : BOOL ;	//TRAVEL DRIVE1 HEALTHY COMMEND
   TRVEL_DRV2_HEALTHY_CMD : BOOL ;	//TRAVEL DRIVE2 HEALTHY COMMEND
   QUNCHING_TIME_POS_PLS : BOOL ;	//QUNCHING TIMER POSITIVE PLUSE BIT
   MAIN_PWR_HEALTHY_BIT : BOOL ;	//MAIN POWER ON HEALTHY BIT
   SPARE1 : INT ;	//SPARE1
   SPARE2 : INT ;	//SPARE2
   SPARE3 : INT ;
   MAX_SPED_LOCO_SET_HW : INT ;	//MAXIMUM SET SPEED FOR LOCO HARDWARE UNSCALING
   MAX_SPED_LOCO_SET_HW1 : INT ;	//MAXIMUM SET SPEED FOR LOCO HARDWARE UNSCALING1
   MAX_SPED_LOCO_SET_HW_REF : REAL ;	//MAXIMUM SET SPEED FOR LOCO HARDWARE SCALING
   MAX_SPED_LOCO_SET_PROFI : INT ;	//MAXIMUM SET SPEED FOR LOCO PROFIBUS UNSCALING
   QUNCHING_SPED_FOR_PROFI : INT ;	//QUNCHING SPEED FOR PROFIBUS MODE
   MAX_SPED_LOCO_PROFI_REF : REAL ;	//MAXIMUM SET SPEED FOR LOCO PROFIBUS SCALING
   SPARE_LOCAL1 : INT ;	//SPARE LOCAL 1
   SPARE_LOCAL2 : INT ;	//SPARE LOCAL 2
   SPARE_LOCAL3 : INT ;	//SPARE LOCAL 3
   SPARE_LOCAL4 : INT ;	//SPARE LOCAL 4
   SPARE_LOCAL5 : INT ;	//SPARE LOCAL 5
   SPARE_LOCAL6 : INT ;	//SPARE LOCAL 6
   SPARE_LOCAL7 : INT ;	//SPARE LOCAL 7
   SPARE_LOCAL8 : INT ;	//SPARE LOCAL 8
   SPARE_LOCAL9 : INT ;	//SPARE LOCAL 9
   SPARE_LOCAL10 : INT ;	//SPARE LOCAL 10
   SPARE_LOCAL11 : INT ;	//SPARE LOCAL 11
   SPARE_LOCAL12 : INT ;	//SPARE LOCAL 12
   FWD_EMER_EMD_LIMIT_SW_FB : BOOL ;	//FORWARD EMERGENCY END LIMIT SWITCH FEED BACK
   REV_EMER_EMD_LIMIT_SW_FB : BOOL ;	//REVERSE EMERGENCY END LIMIT SWITCH FEED BACK
   COMPRSR_BRK_PR_SW_FB : BOOL ;	//COMPRESSOR BRAKE LINE PRESSURE SWITCH FEED BACK
   COMPRSR_MIN_PR_SW_FB : BOOL ;	//COMPRESSOR MINIMUM PRESSURE SWITCH FEED BACK
   QUNCHING_START_PB : BOOL ;	//"QUNCHING_START_PB".
   MANUAL_SELECT_SS : BOOL ;	//MANUAL MODE SELECTON
   AUTO_SELECT_SS : BOOL ;	//AUTO MODE SELECTION
   LAMP_TEST_PB_AT_CD : BOOL ;	//LAMP TEST PB AT CD
   ALARM_ACT_PB_AT_CD : BOOL ;	//ALARM ACCKNOWLODGE PUSH BUTTON PB CD
   TRVL_DRV1_RUNNG_FB : BOOL ;	//TRAVEL DRIVE 1 RUNNING FEED BACK
   TRVL_DRV2_RUNNG_FB : BOOL ;	//TRAVEL DRIVE 2 RUNNING FEED BACK
   SPARE : BOOL ;	//SPARE
   JOY_ST_DEADMAN_BUTTON : BOOL ;	//JOYSTICK DEADMAN BUTTON
   JOY_ST_FWD_POSITN : BOOL ;	//JOYSTICK FORWARD POSITION
   JOY_ST_REV_POSITN : BOOL ;	//JOYSTICK REVERSE POSITION
   JOY_ST_HOME_POSITN : BOOL ;	//JOYSTICK HOME POSITION
   PROFIBUS_HW_SEL_DRV1 : BOOL ;	//PROFIBUS/HARDWARE SELECTION DRIVE 1
   PROFIBUS_HW_SEL_DRV2 : BOOL ;	//PROFIBUS/HARDWARE SELECTION DRIVE 2
   QUNCHING_SLOW_SPED_LS : BOOL ;	//QUNCHING SLOW SPEED LIMIT SWOTCH
   TRVL_DRV1_RDY_STRAT : BOOL ;	//TRAVEL DRIVE 1 READY TO START
   TRVL_DRV1_OLR_TRIP : BOOL ;	//TRAVEL DRIVE 1 OLR TRIP FEED BACK
   TRVL_DRV2_RDY_STRAT : BOOL ;	//TRAVEL DRIVE 2 READY TO START
   TRVL_DRV2_OLR_TRIP : BOOL ;	//TRAVEL DRIVE 2 OLR TRIP FEED BACK
   SPARE_INPUT1 : INT ;	//SPARE INPUT 1
   SPARE_INPUT2 : INT ;	//SPARE INPUT 2
   SPARE_INPUT3 : INT ;	//SPARE INPUT 3
   TRVL_PERMSN_IND : BOOL ;	//TRAVEL PERMISSION INDICATION
   TRVL_DRV1_FWD_CMD : BOOL ;	//TRAVEL DRIVE 1 FORWARD COMMEND
   TRVL_DRV2_FWD_CMD : BOOL ;	//TRAVEL DRIVE 2 FORWARD COMMEND
   TRVL_DRV1_REV_CMD : BOOL ;	//TRAVEL DRIVE 1 REVERSE COMMEND
   TRVL_DRV2_REV_CMD : BOOL ;	//TRAVEL DRIVE 2 REVERSE COMMEND
   AUTO_POSTN_ACK_IND : BOOL ;	//AUTO POSITION ACKNOWLEDGE MENT INDICATION
   JS_SPEED_REF_DI : DINT ;	//JOY STICK SPEED REFERENCE DOUBLE INTEGER
   JS_SPEED_REF_NEG_RMD : INT ;	//JOY STICK SPEED REFERENCE NEGATIVE REMOVED
   JS_SPEED_REF_REAL : REAL ;	//JOY STICK SPEED REFERENCE FLOATING POINT
   SPEED_REF_TO_DRV : INT ;	//SPEED REFERENCE TO DRIVE
   UNSCALING_BLOCK_ERROR : WORD ;	//UN SCALLING BLOCK ERROR
   TR_DRV_1_STATUS_WORD_1 : INT ;	//TRAVEL DRIVE 1 PROFIBUS STATUS WORD 1
   TR_DRV_1_STATUS_WORD_2 : INT ;	//TRAVEL DRIVE 1 PROFIBUS STATUS WORD 2
   TR_DRV_1_STATUS_WORD_3 : INT ;	//TRAVEL DRIVE 1 PROFIBUS STATUS WORD 3
   TR_DRV_1_STATUS_WORD_4 : INT ;	//TRAVEL DRIVE 1 PROFIBUS STATUS WORD 4
   TR_DRV_1_STATUS_WORD_5 : INT ;	//TRAVEL DRIVE 1 PROFIBUS STATUS WORD 5
   TR_DRV_1_STATUS_WORD_6 : INT ;	//TRAVEL DRIVE 1 PROFIBUS STATUS WORD 6
   TR_DRV_1_STATUS_WORD_7 : INT ;	//TRAVEL DRIVE 1 PROFIBUS STATUS WORD 7
   TR_DRV_1_STATUS_WORD_8 : INT ;	//TRAVEL DRIVE 1 PROFIBUS STATUS WORD 8
   TR_DRV_1_STATUS_WORD_9 : INT ;	//TRAVEL DRIVE 1 PROFIBUS STATUS WORD 9
   TR_DRV_1_STATUS_WORD_10 : INT ;	//TRAVEL DRIVE 1 PROFIBUS STATUS WORD 10
   TR_DRV_1_STATUS_WORD_11 : INT ;	//TRAVEL DRIVE 1 PROFIBUS STATUS WORD 11
   TR_DRV_1_STATUS_WORD_12 : INT ;	//TRAVEL DRIVE 1 PROFIBUS STATUS WORD 12
   TR_DRV_1_STATUS_WORD_13 : INT ;	//TRAVEL DRIVE 1 PROFIBUS STATUS WORD 13
   TR_DRV_1_STATUS_WORD_14 : INT ;	//TRAVEL DRIVE 1 PROFIBUS STATUS WORD 14
   TR_DRV_1_STATUS_WORD_15 : INT ;	//TRAVEL DRIVE 1 PROFIBUS STATUS WORD 15
   TR_DRV_1_STATUS_WORD_16 : INT ;	//TRAVEL DRIVE 1 PROFIBUS STATUS WORD 16
   TR_DRV_1_CONTROL_WORD_1 : INT ;	//TRAVEL DRIVE 1 PROFIBUS CONTROL WORD 1
   TR_DRV_1_CONTROL_WORD_2 : INT ;	//TRAVEL DRIVE 1 PROFIBUS CONTROL WORD 2
   TR_DRV_1_CONTROL_WORD_3 : INT ;	//TRAVEL DRIVE 1 PROFIBUS CONTROL WORD 3
   TR_DRV_1_CONTROL_WORD_4 : INT ;	//TRAVEL DRIVE 1 PROFIBUS CONTROL WORD 4
   TR_DRV_1_CONTROL_WORD_5 : INT ;	//TRAVEL DRIVE 1 PROFIBUS CONTROL WORD 5
   TR_DRV_1_CONTROL_WORD_6 : INT ;	//TRAVEL DRIVE 1 PROFIBUS CONTROL WORD 6
   TR_DRV_1_CONTROL_WORD_7 : INT ;	//TRAVEL DRIVE 1 PROFIBUS CONTROL WORD 7
   TR_DRV_1_CONTROL_WORD_8 : INT ;	//TRAVEL DRIVE 1 PROFIBUS CONTROL WORD 8
   TR_DRV_1_CONTROL_WORD_9 : INT ;	//TRAVEL DRIVE 1 PROFIBUS CONTROL WORD 9
   TR_DRV_1_CONTROL_WORD_10 : INT ;	//TRAVEL DRIVE 1 PROFIBUS CONTROL WORD 10
   TR_DRV_1_CONTROL_WORD_11 : INT ;	//TRAVEL DRIVE 1 PROFIBUS CONTROL WORD 11
   TR_DRV_1_CONTROL_WORD_12 : INT ;	//TRAVEL DRIVE 1 PROFIBUS CONTROL WORD 12
   TR_DRV_1_CONTROL_WORD_13 : INT ;	//TRAVEL DRIVE 1 PROFIBUS CONTROL WORD 13
   TR_DRV_1_CONTROL_WORD_14 : INT ;	//TRAVEL DRIVE 1 PROFIBUS CONTROL WORD 14
   TR_DRV_1_CONTROL_WORD_15 : INT ;	//TRAVEL DRIVE 1 PROFIBUS CONTROL WORD 15
   TR_DRV_1_CONTROL_WORD_16 : INT ;	//TRAVEL DRIVE 1 PROFIBUS CONTROL WORD 16
   TR_DRV_1_STAT_WORD_1_ERR : INT ;	//TRAVEL DRIVE 1 DRIVE STATUS WORD 1 READ ERROR
   TR_DRV_1_STAT_WORD_2_ERR : INT ;	//TRAVEL DRIVE 1 DRIVE STATUS WORD 2 READ ERROR
   TR_DRV_1_STAT_WORD_3_ERR : INT ;	//TRAVEL DRIVE 1 DRIVE STATUS WORD 3 READ ERROR
   TR_DRV_1_STAT_WORD_4_ERR : INT ;	//TRAVEL DRIVE 1 DRIVE STATUS WORD 4 READ ERROR
   TR_DRV_1_CTRL_WORD_1_ERR : INT ;	//TRAVEL DRIVE 1 DRIVE CONTROL WORD 1 WRITE ERROR
   TR_DRV_1_CTRL_WORD_2_ERR : INT ;	//TRAVEL DRIVE 1 DRIVE CONTROL WORD 2 WRITE ERROR
   TR_DRV_1_CTRL_WORD_3_ERR : INT ;	//TRAVEL DRIVE 1 DRIVE CONTROL WORD 3 WRITE ERROR
   TR_DRV_1_CTRL_WORD_4_ERR : INT ;	//TRAVEL DRIVE 1 DRIVE CONTROL WORD 4 WRITE ERROR
   TR_DRV_2_STATUS_WORD_1 : INT ;	//TRAVEL DRIVE 2 PROFIBUS STATUS WORD 1
   TR_DRV_2_STATUS_WORD_2 : INT ;	//TRAVEL DRIVE 2 PROFIBUS STATUS WORD 2
   TR_DRV_2_STATUS_WORD_3 : INT ;	//TRAVEL DRIVE 2 PROFIBUS STATUS WORD 3
   TR_DRV_2_STATUS_WORD_4 : INT ;	//TRAVEL DRIVE 2 PROFIBUS STATUS WORD 4
   TR_DRV_2_STATUS_WORD_5 : INT ;	//TRAVEL DRIVE 2 PROFIBUS STATUS WORD 5
   TR_DRV_2_STATUS_WORD_6 : INT ;	//TRAVEL DRIVE 2 PROFIBUS STATUS WORD 6
   TR_DRV_2_STATUS_WORD_7 : INT ;	//TRAVEL DRIVE 2 PROFIBUS STATUS WORD 7
   TR_DRV_2_STATUS_WORD_8 : INT ;	//TRAVEL DRIVE 2 PROFIBUS STATUS WORD 8
   TR_DRV_2_STATUS_WORD_9 : INT ;	//TRAVEL DRIVE 2 PROFIBUS STATUS WORD 9
   TR_DRV_2_STATUS_WORD_10 : INT ;	//TRAVEL DRIVE 2 PROFIBUS STATUS WORD 10
   TR_DRV_2_STATUS_WORD_11 : INT ;	//TRAVEL DRIVE 2 PROFIBUS STATUS WORD 11
   TR_DRV_2_STATUS_WORD_12 : INT ;	//TRAVEL DRIVE 2 PROFIBUS STATUS WORD 12
   TR_DRV_2_STATUS_WORD_13 : INT ;	//TRAVEL DRIVE 2 PROFIBUS STATUS WORD 13
   TR_DRV_2_STATUS_WORD_14 : INT ;	//TRAVEL DRIVE 2 PROFIBUS STATUS WORD 14
   TR_DRV_2_STATUS_WORD_15 : INT ;	//TRAVEL DRIVE 2 PROFIBUS STATUS WORD 15
   TR_DRV_2_STATUS_WORD_16 : INT ;	//TRAVEL DRIVE 2 PROFIBUS STATUS WORD 16
   TR_DRV_2_CONTROL_WORD_1 : INT ;	//TRAVEL DRIVE 2 PROFIBUS CONTROL WORD 1
   TR_DRV_2_CONTROL_WORD_2 : INT ;	//TRAVEL DRIVE 2 PROFIBUS CONTROL WORD 2
   TR_DRV_2_CONTROL_WORD_3 : INT ;	//TRAVEL DRIVE 2 PROFIBUS CONTROL WORD 3
   TR_DRV_2_CONTROL_WORD_4 : INT ;	//TRAVEL DRIVE 2 PROFIBUS CONTROL WORD 4
   TR_DRV_2_CONTROL_WORD_5 : INT ;	//TRAVEL DRIVE 2 PROFIBUS CONTROL WORD 5
   TR_DRV_2_CONTROL_WORD_6 : INT ;	//TRAVEL DRIVE 2 PROFIBUS CONTROL WORD 6
   TR_DRV_2_CONTROL_WORD_7 : INT ;	//TRAVEL DRIVE 2 PROFIBUS CONTROL WORD 7
   TR_DRV_2_CONTROL_WORD_8 : INT ;	//TRAVEL DRIVE 2 PROFIBUS CONTROL WORD 8
   TR_DRV_2_CONTROL_WORD_9 : INT ;	//TRAVEL DRIVE 2 PROFIBUS CONTROL WORD 9
   TR_DRV_2_CONTROL_WORD_10 : INT ;	//TRAVEL DRIVE 2 PROFIBUS CONTROL WORD 10
   TR_DRV_2_CONTROL_WORD_11 : INT ;	//TRAVEL DRIVE 2 PROFIBUS CONTROL WORD 11
   TR_DRV_2_CONTROL_WORD_12 : INT ;	//TRAVEL DRIVE 2 PROFIBUS CONTROL WORD 12
   TR_DRV_2_CONTROL_WORD_13 : INT ;	//TRAVEL DRIVE 2 PROFIBUS CONTROL WORD 13
   TR_DRV_2_CONTROL_WORD_14 : INT ;	//TRAVEL DRIVE 2 PROFIBUS CONTROL WORD 14
   TR_DRV_2_CONTROL_WORD_15 : INT ;	//TRAVEL DRIVE 2 PROFIBUS CONTROL WORD 15
   TR_DRV_2_CONTROL_WORD_16 : INT ;	//TRAVEL DRIVE 2 PROFIBUS CONTROL WORD 16
   TR_DRV_2_STAT_WORD_1_ERR : INT ;	//TRAVEL DRIVE 2 DRIVE STATUS WORD 1 READ ERROR
   TR_DRV_2_STAT_WORD_2_ERR : INT ;	//TRAVEL DRIVE 2 DRIVE STATUS WORD 2 READ ERROR
   TR_DRV_2_STAT_WORD_3_ERR : INT ;	//TRAVEL DRIVE 2 DRIVE STATUS WORD 3 READ ERROR
   TR_DRV_2_STAT_WORD_4_ERR : INT ;	//TRAVEL DRIVE 2 DRIVE STATUS WORD 4 READ ERROR
   TR_DRV_2_CTRL_WORD_1_ERR : INT ;	//TRAVEL DRIVE 2 DRIVE CONTROL WORD 1 WRITE ERROR
   TR_DRV_2_CTRL_WORD_2_ERR : INT ;	//TRAVEL DRIVE 2 DRIVE CONTROL WORD 2 WRITE ERROR
   TR_DRV_2_CTRL_WORD_3_ERR : INT ;	//TRAVEL DRIVE 2 DRIVE CONTROL WORD 3 WRITE ERROR
   TR_DRV_2_CTRL_WORD_4_ERR : INT ;	//TRAVEL DRIVE 2 DRIVE CONTROL WORD 4 WRITE ERROR
   DR_1_CW_B0_RDY_TO_OPER : BOOL ;	//TRAVEL DRIVE 1 CONTROL WORD BIT 0 - READY TO OPERATE - OFF1 - PROFIBUS
   DR_1_CW_B1_OFF_2 : BOOL ;	//TRAVEL DRIVE 1 CONTROL WORD BIT 1 - OFF2 - PROFIBUS
   DR_1_CW_B2_OFF_3 : BOOL ;	//TRAVEL DRIVE 1 CONTROL WORD BIT 2 - OFF3 - PROFIBUS
   DR_1_CW_B3_OPER_ENAB : BOOL ;	//TRAVEL DRIVE 1 CONTROL WORD BIT 3 - OPERATION ENABLE - PROFIBUS
   DR_1_CW_B4_RMP_OUT_ZERO : BOOL ;	//TRAVEL DRIVE 1 CONTROL WORD BIT 4 - RAMP OUT ZERO - PROFIBUS
   DR_1_CW_B5_RMP_HLD : BOOL ;	//TRAVEL DRIVE 1 CONTROL WORD BIT 5 - RAMP HOLD - PROFIBUS
   DR_1_CW_B6_RMP_IN_ZERO : BOOL ;	//TRAVEL DRIVE 1 CONTROL WORD BIT 6 - RAMP IN ZERO - PROFIBUS
   DR_1_CW_B7_FLT_RST : BOOL ;	//TRAVEL DRIVE 1 CONTROL WORD BIT 7 - FAULT RESET - PROFIBUS
   DR_1_CW_B8_INCH_1 : BOOL ;	//TRAVEL DRIVE 1 CONTROL WORD BIT 8 - INCHING 1 - PROFIBUS
   DR_1_CW_B9_INCH_2 : BOOL ;	//TRAVEL DRIVE 1 CONTROL WORD BIT 9 - INCHING 2 - PROFIBUS
   DR_1_CW_B10_RMT_CMD : BOOL ;	//TRAVEL DRIVE 1 CONTROL WORD BIT 10 - REMOTE COMMAND - PROFIBUS
   DR_1_CW_B11 : BOOL ;	//TRAVEL DRIVE 1 CONTROL WORD BIT 11 - DRIVE SPECIFIC - PROFOBUS
   DR_1_CW_B12 : BOOL ;	//TRAVEL DRIVE 1 CONTROL WORD BIT 12 - DRIVE SPECIFIC - PROFOBUS
   DR_1_CW_B13 : BOOL ;	//TRAVEL DRIVE 1 CONTROL WORD BIT 13 - DRIVE SPECIFIC - PROFOBUS
   DR_1_CW_B14 : BOOL ;	//TRAVEL DRIVE 1 CONTROL WORD BIT 14 - DRIVE SPECIFIC - PROFOBUS
   DR_1_CW_B15 : BOOL ;	//TRAVEL DRIVE 1 CONTROL WORD BIT 15 - DRIVE SPECIFIC - PROFOBUS
   DR_1_SW_B0_RDY_ON : BOOL ;	//TRAVEL DRIVE 1 STATUS WORD BIT 0 - READY TO OPERATE - OFF1 - PROFIBUS
   DR_1_SW_B1_RDY_TO_OPER : BOOL ;	//TRAVEL DRIVE 1 STATUS WORD BIT 1 - REDY TO OPERATE - PROFIBUS
   DR_1_SW_B2_REF_RDY : BOOL ;	//TRAVEL DRIVE 1 STATUS WORD BIT 2 - ENABEL OPERATION - PROFIBUS
   DR_1_SW_B3_TRIPPED : BOOL ;	//TRAVEL DRIVE 1 STATUS WORD BIT 3 - FAULT - PROFIBUS
   DR_1_SW_B4_OFF_2_STA : BOOL ;	//TRAVEL DRIVE 1 STATUS WORD BIT 4 - OFF 2 STATUS - PROFIBUS
   DR_1_SW_B5_OFF_3_STA : BOOL ;	//TRAVEL DRIVE 1 STATUS WORD BIT 5 - OFF 3 STATUS - PROFIBUS
   DR_1_SW_B6_SWC_ON_INHB : BOOL ;	//TRAVEL DRIVE 1 STATUS WORD BIT 6 - SWITCH ON INHIBIT - PROFIBUS
   DR_1_SW_B7_ALARM : BOOL ;	//TRAVEL DRIVE 1 STATUS WORD BIT 7 - WARNING/ALARM - PROFIBUS
   DR_1_SW_B8_AT_SETPOINT : BOOL ;	//TRAVEL DRIVE 1 STATUS WORD BIT 8 - OPERATING - PROFIBUS
   DR_1_SW_B9_REMOTE : BOOL ;	//TRAVEL DRIVE 1 STATUS WORD BIT 9 - DRIVE CONTROL REMOTE\LOCAL - PROFIBUS
   DR_1_SW_B10_ABOVE_LIMIT : BOOL ;	//TRAVEL DRIVE 1 STATUS WORD BIT 10 - SPEED ABOVE LIMIT - PROFIBUS
   DR_1_SW_B11 : BOOL ;	//TRAVEL DRIVE 1 STATUS WORD BIT 11 - DRIVE SPECIFIC - PROFOBUS
   DR_1_SW_B12 : BOOL ;	//TRAVEL DRIVE 1 STATUS WORD BIT 12 - DRIVE SPECIFIC - PROFOBUS
   DR_1_SW_B13 : BOOL ;	//TRAVEL DRIVE 1 STATUS WORD BIT 13 - DRIVE SPECIFIC - PROFOBUS
   DR_1_SW_B14 : BOOL ;	//TRAVEL DRIVE 1 STATUS WORD BIT 14 - DRIVE SPECIFIC - PROFOBUS
   DR_1_SW_B15 : BOOL ;	//TRAVEL DRIVE 1 STATUS WORD BIT 15 - DRIVE SPECIFIC - PROFOBUS
   JS_SPD_REF_DI_PF : DINT ;	//JOY STICK SPEED REFERENCE IN DOUBLE INTEGER
   JS_SPD_REF_REAL_PF : REAL ;	//JOY STICK SPEED REFERENCE IN REAL(FLOATING POINT)
   JS_SPD_REF_UN_SL_FLT_PF : WORD ;	//JOY STICK SPEED REFERENCE UNSCALLING FAULT
   TRA_SPD_REF_VAL_PF : INT ;	//TRAVEL SPEED REFERENCE VALUE
   DR_2_CW_B0_RDY_TO_OPER : BOOL ;	//TRAVEL DRIVE 2 CONTROL WORD BIT 0 - READY TO OPERATE - OFF1 - PROFIBUS
   DR_2_CW_B1_OFF_2 : BOOL ;	//TRAVEL DRIVE 2 CONTROL WORD BIT 1 - OFF2 - PROFIBUS
   DR_2_CW_B2_OFF_3 : BOOL ;	//TRAVEL DRIVE 2 CONTROL WORD BIT 2 - OFF3 - PROFIBUS
   DR_2_CW_B3_OPER_ENAB : BOOL ;	//TRAVEL DRIVE 2 CONTROL WORD BIT 3 - OPERATION ENABLE - PROFIBUS
   DR_2_CW_B4_RMP_OUT_ZERO : BOOL ;	//TRAVEL DRIVE 2 CONTROL WORD BIT 4 - RAMP OUT ZERO - PROFIBUS
   DR_2_CW_B5_RMP_HLD : BOOL ;	//TRAVEL DRIVE 2 CONTROL WORD BIT 5 - RAMP HOLD - PROFIBUS
   DR_2_CW_B6_RMP_IN_ZERO : BOOL ;	//TRAVEL DRIVE 2 CONTROL WORD BIT 6 - RAMP IN ZERO - PROFIBUS
   DR_2_CW_B7_FLT_RST : BOOL ;	//TRAVEL DRIVE 2 CONTROL WORD BIT 7 - FAULT RESET - PROFIBUS
   DR_2_CW_B8_INCH_1 : BOOL ;	//TRAVEL DRIVE 2 CONTROL WORD BIT 8 - INCHING 1 - PROFIBUS
   DR_2_CW_B9_INCH_2 : BOOL ;	//TRAVEL DRIVE 2 CONTROL WORD BIT 9 - INCHING 2 - PROFIBUS
   DR_2_CW_B10_RMT_CMD : BOOL ;	//TRAVEL DRIVE 2 CONTROL WORD BIT 10 - REMOTE COMMAND - PROFIBUS
   DR_2_CW_B11 : BOOL ;	//TRAVEL DRIVE 2 CONTROL WORD BIT 11 - DRIVE SPECIFIC - PROFOBUS
   DR_2_CW_B12 : BOOL ;	//TRAVEL DRIVE 2 CONTROL WORD BIT 12 - DRIVE SPECIFIC - PROFOBUS
   DR_2_CW_B13 : BOOL ;	//TRAVEL DRIVE 2 CONTROL WORD BIT 13 - DRIVE SPECIFIC - PROFOBUS
   DR_2_CW_B14 : BOOL ;	//TRAVEL DRIVE 2 CONTROL WORD BIT 14 - DRIVE SPECIFIC - PROFOBUS
   DR_2_CW_B15 : BOOL ;	//TRAVEL DRIVE 2 CONTROL WORD BIT 15 - DRIVE SPECIFIC - PROFOBUS
   DR_2_SW_B0_RDY_ON : BOOL ;	//TRAVEL DRIVE 2 STATUS WORD BIT 0 - READY TO OPERATE - OFF1 - PROFIBUS
   DR_2_SW_B1_RDY_TO_OPER : BOOL ;	//TRAVEL DRIVE 2 STATUS WORD BIT 1 - REDY TO OPERATE - PROFIBUS
   DR_2_SW_B2_REF_RDY : BOOL ;	//TRAVEL DRIVE 2 STATUS WORD BIT 2 - ENABEL OPERATION - PROFIBUS
   DR_2_SW_B3_TRIPPED : BOOL ;	//TRAVEL DRIVE 2 STATUS WORD BIT 3 - FAULT - PROFIBUS
   DR_2_SW_B4_OFF_2_STA : BOOL ;	//TRAVEL DRIVE 2 STATUS WORD BIT 4 - OFF 2 STATUS - PROFIBUS
   DR_2_SW_B5_OFF_3_STA : BOOL ;	//TRAVEL DRIVE 2 STATUS WORD BIT 5 - OFF 3 STATUS - PROFIBUS
   DR_2_SW_B6_SWC_ON_INHB : BOOL ;	//TRAVEL DRIVE 2 STATUS WORD BIT 6 - SWITCH ON INHIBIT - PROFIBUS
   DR_2_SW_B7_ALARM : BOOL ;	//TRAVEL DRIVE 2 STATUS WORD BIT 7 - WARNING/ALARM - PROFIBUS
   DR_2_SW_B8_AT_SETPOINT : BOOL ;	//TRAVEL DRIVE 2 STATUS WORD BIT 8 - OPERATING - PROFIBUS
   DR_2_SW_B9_REMOTE : BOOL ;	//TRAVEL DRIVE 2 STATUS WORD BIT 9 - DRIVE CONTROL REMOTE\LOCAL - PROFIBUS
   DR_2_SW_B10_ABOVE_LIMIT : BOOL ;	//TRAVEL DRIVE 2 STATUS WORD BIT 10 - SPEED ABOVE LIMIT - PROFIBUS
   DR_2_SW_B11 : BOOL ;	//TRAVEL DRIVE 2 STATUS WORD BIT 11 - DRIVE SPECIFIC - PROFOBUS
   DR_2_SW_B12 : BOOL ;	//TRAVEL DRIVE 2 STATUS WORD BIT 12 - DRIVE SPECIFIC - PROFOBUS
   DR_2_SW_B13 : BOOL ;	//TRAVEL DRIVE 2 STATUS WORD BIT 13 - DRIVE SPECIFIC - PROFOBUS
   DR_2_SW_B14 : BOOL ;	//TRAVEL DRIVE 2 STATUS WORD BIT 14 - DRIVE SPECIFIC - PROFOBUS
   DR_2_SW_B15 : BOOL ;	//TRAVEL DRIVE 2 STATUS WORD BIT 15 - DRIVE SPECIFIC - PROFOBUS
   DR_1_ACT_SPD_PF : REAL ;	//TRAVEL DRIVE 1 ACTUAL SPEED - PROFIBUS
   DR_1_ACT_SPD_SCL_ERR : WORD ;	//TRAVEL DRIVE 1 ACTUAL SPEED SCALING ERROR - PROFIBUS
   DR_2_ACT_SPD_PF : REAL ;	//TRAVEL DRIVE 2 ACTUAL SPEED - PROFIBUS
   DR_2_ACT_SPD_SCL_ERR : WORD ;	//TRAVEL DRIVE 2 ACTUAL SPEED SCALING ERROR - PROFIBUS
   TRA_FWD_CHNG_OVR_DEL : BOOL ;	//TRAVEL DRIVE FORWARD CHANGE OVER DELAY
   TRA_REV_CHNG_OVR_DEL : BOOL ;	//TRAVEL DRIVE REVERSE CHANGE OVER DELAY
   TRVEL_DRV1_FWD_CMD_PF : BOOL ;	//TRAVEL DRIVE1 FORWARD COMMEND PROFIBUS
   TRVEL_DRV1_REV_CMD_PF : BOOL ;	//TRAVEL DRIVE1 REVERSE COMMEND PROFIBUS
   TRVEL_DRV2_FWD_CMD_PF : BOOL ;	//TRAVEL DRIVE12 FORWARD COMMEND PROFIBUS
   TRVEL_DRV2_REV_CMD_PF : BOOL ;	//TRAVEL DRIVE2 REVERSE COMMEND PROFIBUS
   PULSE_1 : BOOL ;	//PULSE 1
   PULSE_2 : BOOL ;	//PULSE 2
   PULSE_3 : BOOL ;	//PULSE 3
   PULSE_4 : BOOL ;	//PULSE 4
   DRIVE_1_ISU_CHARGE : BOOL ;	//TRAVEL DRIVE 1 ISU CHARGE
   DRIVE_2_ISU_CHARGE : BOOL ;	//TRAVEL DRIVE 1 ISU CHARGE
   DRV_1_ISU_CHARGE_CMD : BOOL ;	//DRIVE 1 ISU CHARGE COMMAND
   DRV_2_ISU_CHARGE_CMD : BOOL ;	//DRIVE 2 ISU CHARGE COMMAND
   CRIP_SPEED : BOOL ;	//CRIPPING SPEED
   DRV_1_ISU_CMD : BOOL ;	//TRAVEL DRIVE 1 ISU COMMAND
   DRV_2_ISU_CMD : BOOL ;	//TRAVEL DRIVE 2 ISU COMMAND
   HOOTER_ON_CMD : BOOL ;	//HOOTER ON COMMAND
   LIGHT_ON_CMD : BOOL ;	//LIGHT ON COMMAND
  END_STRUCT ;	
BEGIN
END_DATA_BLOCK

DATA_BLOCK "COMMON_DB"	// DB 4
VERSION : 0.1
  STRUCT
   EMER_PRESSED : BOOL ;	//EMERGENCY PRESSED
   ONE_SEC_PLS_TIME_BIT : BOOL ;	//ONE SECOND PLUSE TIMER BIT
   TWO_SEC_PLS_TIME_BIT : BOOL ;	//TWO SECOND PLUSE TIMER BIT
   ONE_SEC_PLS_BIT1 : BOOL ;	//ONE SECOND PLUSE BIT1
   ONE_SEC_POS_BIT : BOOL ;	//ONE SECOND POSITIVE PLUSE BIT
   SPARE1 : INT ;	//SPARE1
   SPARE2 : INT ;	//SPARE2
   SPARE3 : INT ;	//SPARE3
   SPARE4 : INT ;	//SPARE4
   TIME_CONT_DELAY_500MS : INT ;	//500 MS TIMER COUNT DELAY
  END_STRUCT ;	
BEGIN
END_DATA_BLOCK

DATA_BLOCK "TATA_COMMUNICATION_DB"	// DB 5
AUTHOR : Kamillas
VERSION : 0.1
  STRUCT
   PULSE_1 : BOOL ;	//PULSE 1
   PULSE_2 : BOOL ;	//PULSE 2
   PULSE_3 : BOOL ;	//PULSE 3
   PULSE_4 : BOOL ;	//PULSE 4
   TATA_DATA_READ_ERROR : INT ;	//TATA PLC DATA READ ERROR
   TATA_DATA_WRITE_ERROR : INT ;	//TATA PLC DATA WRITE ERROR
  END_STRUCT ;	
BEGIN
END_DATA_BLOCK

DATA_BLOCK "WinCC_Interface_DB"	// DB 6
VERSION : 0.1
  STRUCT
   STAT0 : BOOL ;
   LAMP_TEST : BOOL ;	//LAMP TEST
   ALARM_ACK : BOOL ;	//ALARM ACK
   TRAVEL_MANUAL_SEL : BOOL ;	//TRAVEL MANUAL MODE SEL
   TRAVEL_AUTO_SEL : BOOL ;	//TRAVEL AUTO MODE SEL
   SPARE : BOOL ;	//SPARE
   EMG_STOP_PB : BOOL ;	//EMERGENCY STOP PB
   COMP_SELE : BOOL ;	//COMPRESSOR 2 SEL
   CMPR1_START : BOOL ;	//COMPRESSOR 1 START PB
   CMPR1_STOP : BOOL ;	//COMPRESSOR 1 STOP PB
   CMPR2_START : BOOL ;	//COMPRESSOR 2 START PB
   CMPR2_STOP : BOOL ;	//COMPRESSOR 2 STOP PB
   TRAVEL_CREEPING_SPEED : BOOL ;	//CREEPING SPEED
   STAT13 : BOOL ;
   STAT14 : BOOL ;
   STAT15 : BOOL ;
   COMPR_SELECT_TAG : BOOL ;
   STAT17 : BOOL ;
   STAT18 : BOOL ;
   STAT19 : BOOL ;
   STAT20 : BOOL ;
   STAT21 : BOOL ;
   STAT22 : BOOL ;
   STAT23 : BOOL ;
   TRAVEL_SELECT_TAG : BOOL ;
   STAT25 : BOOL ;
   STAT26 : BOOL ;
   STAT27 : BOOL ;
   STAT28 : BOOL ;
   STAT29 : BOOL ;
   STAT30 : BOOL ;
   STAT31 : BOOL ;
   CRIP_SPD_TRA_TAG : BOOL ;
   STAT33 : BOOL ;
   STAT34 : BOOL ;
   STAT35 : BOOL ;
   STAT36 : BOOL ;
   STAT37 : BOOL ;
   STAT38 : BOOL ;
   STAT39 : BOOL ;
   STAT40 : BOOL ;
   STAT41 : BOOL ;
   STAT42 : BOOL ;
   STAT43 : BOOL ;
   STAT44 : BOOL ;
   STAT45 : BOOL ;
   STAT46 : BOOL ;
   STAT47 : BOOL ;
   STAT48 : BOOL ;
   STAT49 : BOOL ;
   STAT50 : BOOL ;
   STAT51 : BOOL ;
   STAT52 : BOOL ;
   STAT53 : BOOL ;
   STAT54 : BOOL ;
   STAT55 : BOOL ;
   STAT56 : BOOL ;
   STAT57 : BOOL ;
   STAT58 : BOOL ;
   STAT59 : BOOL ;
   STAT60 : BOOL ;
   STAT61 : BOOL ;
   STAT62 : BOOL ;
   STAT63 : BOOL ;
   STAT64 : BOOL ;
   STAT65 : BOOL ;
   STAT66 : BOOL ;
   STAT67 : BOOL ;
   STAT68 : BOOL ;
   STAT69 : BOOL ;
   STAT70 : BOOL ;
   STAT71 : BOOL ;
   STAT72 : BOOL ;
   STAT73 : BOOL ;
   STAT74 : BOOL ;
   STAT75 : BOOL ;
   STAT76 : BOOL ;
   STAT77 : BOOL ;
   STAT78 : BOOL ;
   STAT79 : BOOL ;
   STAT80 : BOOL ;
   STAT81 : BOOL ;
   STAT82 : BOOL ;
   STAT83 : BOOL ;
   STAT84 : BOOL ;
   STAT85 : BOOL ;
   STAT86 : BOOL ;
   STAT87 : BOOL ;
   STAT88 : BOOL ;
   STAT89 : BOOL ;
   STAT90 : BOOL ;
   STAT91 : BOOL ;
   STAT92 : BOOL ;
   STAT93 : BOOL ;
   STAT94 : BOOL ;
   STAT95 : BOOL ;
   STAT96 : BOOL ;
   STAT97 : BOOL ;
   STAT98 : BOOL ;
   STAT99 : BOOL ;
   STAT100 : BOOL ;
   STAT101 : BOOL ;
   STAT102 : BOOL ;
   STAT103 : BOOL ;
   STAT104 : BOOL ;
   STAT105 : BOOL ;
   STAT106 : BOOL ;
   STAT107 : BOOL ;
   STAT108 : BOOL ;
   STAT109 : BOOL ;
   STAT110 : BOOL ;
   STAT111 : BOOL ;
   STAT112 : BOOL ;
   STAT113 : BOOL ;
   STAT114 : BOOL ;
   STAT115 : BOOL ;
   STAT116 : BOOL ;
   STAT117 : BOOL ;
   STAT118 : BOOL ;
   STAT119 : BOOL ;
   STAT120 : BOOL ;
   STAT121 : BOOL ;
   STAT122 : BOOL ;
   STAT123 : BOOL ;
   STAT124 : BOOL ;
   STAT125 : BOOL ;
   STAT126 : BOOL ;
   STAT127 : BOOL ;
   STAT128 : BOOL ;
   STAT129 : BOOL ;
   STAT130 : BOOL ;
   STAT131 : BOOL ;
   STAT132 : BOOL ;
   STAT133 : BOOL ;
   STAT134 : BOOL ;
   STAT135 : BOOL ;
   STAT136 : BOOL ;
   STAT137 : BOOL ;
   STAT138 : BOOL ;
   STAT139 : BOOL ;
   STAT140 : BOOL ;
   STAT141 : BOOL ;
   STAT142 : BOOL ;
   STAT143 : BOOL ;
   STAT144 : BOOL ;
   STAT145 : BOOL ;
   STAT146 : BOOL ;
   STAT147 : BOOL ;
   STAT148 : BOOL ;
   STAT149 : BOOL ;
   STAT150 : BOOL ;
   STAT151 : BOOL ;
   STAT152 : BOOL ;
   STAT153 : BOOL ;
   STAT154 : BOOL ;
   STAT155 : BOOL ;
   STAT156 : BOOL ;
   STAT157 : BOOL ;
   STAT158 : BOOL ;
   STAT159 : BOOL ;
   STAT160 : BOOL ;
   STAT161 : BOOL ;
   STAT162 : BOOL ;
   STAT163 : BOOL ;
   STAT164 : BOOL ;
   STAT165 : BOOL ;
   STAT166 : BOOL ;
   STAT167 : BOOL ;
   STAT168 : BOOL ;
   STAT169 : BOOL ;
   STAT170 : BOOL ;
   STAT171 : BOOL ;
   STAT172 : BOOL ;
   STAT173 : BOOL ;
   STAT174 : BOOL ;
   STAT175 : BOOL ;
   STAT176 : BOOL ;
   STAT177 : BOOL ;
   STAT178 : BOOL ;
   STAT179 : BOOL ;
   STAT180 : BOOL ;
   STAT181 : BOOL ;
   STAT182 : BOOL ;
   STAT183 : BOOL ;
   STAT184 : BOOL ;
   STAT185 : BOOL ;
   STAT186 : BOOL ;
   STAT187 : BOOL ;
   STAT188 : BOOL ;
   STAT189 : BOOL ;
   STAT190 : BOOL ;
   STAT191 : BOOL ;
   STAT192 : BOOL ;
   STAT193 : BOOL ;
   STAT194 : BOOL ;
   STAT195 : BOOL ;
   STAT196 : BOOL ;
   STAT197 : BOOL ;
   STAT198 : BOOL ;
   STAT199 : BOOL ;
   STAT200 : BOOL ;
   STAT201 : BOOL ;
   STAT202 : BOOL ;
   STAT203 : BOOL ;
   STAT204 : BOOL ;
   STAT205 : BOOL ;
   STAT206 : BOOL ;
   STAT207 : BOOL ;
   STAT208 : BOOL ;
   STAT209 : BOOL ;
   STAT210 : BOOL ;
   STAT211 : BOOL ;
   STAT212 : BOOL ;
   STAT213 : BOOL ;
   STAT214 : BOOL ;
   STAT215 : BOOL ;
   STAT216 : BOOL ;
   STAT217 : BOOL ;
   STAT218 : BOOL ;
   STAT219 : BOOL ;
   STAT220 : BOOL ;
   STAT221 : BOOL ;
   STAT222 : BOOL ;
   STAT223 : BOOL ;
   STAT224 : BOOL ;
   STAT225 : BOOL ;
   STAT226 : BOOL ;
   STAT227 : BOOL ;
   STAT228 : BOOL ;
   STAT229 : BOOL ;
   STAT230 : BOOL ;
   STAT231 : BOOL ;
   COMP_SEL : BOOL ;
   A : BOOL ;
   A1 : BOOL ;
   A2 : BOOL ;
   A3 : BOOL ;
   A4 : BOOL ;
   A5 : BOOL ;
   A6 : BOOL ;
   EMER : BOOL ;
  END_STRUCT ;	
BEGIN
END_DATA_BLOCK

DATA_BLOCK "POWER_ON_DB"	// DB 7
VERSION : 0.1
  STRUCT
   MAIN_PWR_ON_IND_BIT : BOOL ;	//MAIN OWER ON INDICATION BIT
   MAIN_PWR_HEALTHY_BIT : BOOL ;	//MAIN POWER ON HEALTHY BIT
   MAIN_PWR_ON_CMD_BIT : BOOL ;	//MAIN POWER ON COMMEND BIT
   MAIN_PWR_START_CMD : BOOL ;	//MAIN_POWER_START COMMEND
   MAIN_CNTRL_PWR_ON_IND : BOOL ;	//MAIN POWER CONTROL ON COMMEND
   MAIN_PWR_START_POS_PLS : BOOL ;	//MAIN_POWER_START POSITIVE PLUSE
   MAIN_PWR_ON_POS_PLS : BOOL ;	//MAIN OWER ON POSITIVE PLUSE BIT
   ONE_SEC_PLS_BIT : BOOL ;	//ONE SECOND PLUSE BIT
   SPARE_LOCAL1 : INT ;	//SPARE LOCAL 1
   SPARE_LOCAL2 : INT ;	//SPARE LOCAL 2
   SPARE_LOCAL3 : INT ;	//SPARE LOCAL 3
   SPARE_LOCAL4 : INT ;	//SPARE LOCAL 4
   SPARE_LOCAL5 : DINT ;	//SPARE LOCAL 5
   SPARE_LOCAL6 : DINT ;	//SPARE LOCAL 6
   SPARE_LOCAL7 : DINT ;	//SPARE LOCAL 7
   SPARE_LOCAL8 : DINT ;	//SPARE LOCAL 8
   SPARE_LOCAL9 : DINT ;	//SPARE LOCAL 9
   SPARE_LOCAL10 : DINT ;	//SPARE LOCAL 10
   SPARE_LOCAL11 : DINT ;	//SPARE LOCAL 11
   SPARE_LOCAL12 : DINT ;	//SPARE LOCAL 12
   SPARE_LOCAL13 : DINT ;	//SPARE LOCAL 13
   SPARE_LOCAL14 : DINT ;	//SPARE LOCAL 14
   EMER_PRESSED_POWER_ON : BOOL ;	//EMERGENCY PRESSED FOR POWER ON CONDITION
   FWD_EMER_END_LIMIT_SW_FB : BOOL ;	//FORWARD EMERGENCY END LIMIT SWITCH FEED BACK
   REV_EMER_END_LIMIT_SW_FB : BOOL ;	//REVERSE EMERGENCY END LIMIT SWITCH FEED BACK
   MAIN_RUNING_FB : BOOL ;	//MAIN POWER RUNNING FEED BACK
   ALARM_ACT_PB_CD : BOOL ;	//ALARM ACKNOWLEDGE PUSH BUTTON AT CD
   CONTROL_PWR_ON_FB : BOOL ;	//CONTROL POWER ON FEED BACK
   LAMP_TEST_PB_AT_CD : BOOL ;	//LAMP TEST PUSH BUTTON AT CD
   SPARE_INPUT1 : INT ;	//SPARE INPUT 1
   SPARE_INPUT2 : INT ;	//SPARE INPUT 2
   SPARE_INPUT3 : INT ;	//SPARE INPUT 3
   SPARE_INPUT4 : INT ;	//SPARE INPUT 4
   MAIN_PWR_START_CMD1 : BOOL ;	//MAIN POWER START COMMEND
   CONTROL_ON_IND : BOOL ;	//CONTROL POWER ON INDICATION
  END_STRUCT ;	
BEGIN
END_DATA_BLOCK

DATA_BLOCK "ACTUAL_TIME_DB"	// DB 8
VERSION : 0.1
BEGIN
// 400 bytes; values not shown
END_DATA_BLOCK

DATA_BLOCK "COMPRESSOR_DB"	// DB 9
VERSION : 0.1
  STRUCT
   COMPRSR_INTLCK_BIT : BOOL ;	//COMPRESSOR INTERLOCKS BIT
   COMPRSR_1_ON_CMD_BIT : BOOL ;	//COMPRESSOR 1 ON COMMEND BIT
   COMPRSR_2_ON_CMD_BIT : BOOL ;	//COMPRESSOR 2 ON COMMEND BIT
   COMPRSR_1_ON_IND_BIT : BOOL ;	//COMPRESSOR 1 ON INDICATION BIT
   COMPRSR_2_ON_IND_BIT : BOOL ;	//COMPRESSOR 2 ON INDICATION BIT
   COMPRSR_1_POS_PLS : BOOL ;	//COMPRESSOR 1 POSITIVE PLUSE BIT
   COMPRSR_2_POS_PLS : BOOL ;	//COMPRESSOR 2 POSITIVE PLUSE BIT
   MAIN_PWR_HEALTHY_BIT : BOOL ;	//MAIN POWER ON HEALTHY BIT
   SPARE_LOCAL1 : INT ;	//SPRE LOCAL MEMORY1
   SPARE_LOCAL2 : INT ;	//SPRE LOCAL MEMORY12
   SPARE_LOCAL3 : INT ;	//SPRE LOCAL MEMORY3
   SPARE_LOCAL4 : INT ;	//SPRE LOCAL MEMORY4
   SPARE_LOCAL5 : DINT ;	//SPRE LOCAL MEMORY5
   SPARE_LOCAL6 : DINT ;	//SPRE LOCAL MEMORY6
   SPARE_LOCAL7 : DINT ;	//SPRE LOCAL MEMORY7
   SPARE_LOCAL8 : DINT ;	//SPRE LOCAL MEMORY8
   SPARE_LOCAL9 : DINT ;	//SPRE LOCAL MEMORY9
   SPARE_LOCAL10 : DINT ;	//SPRE LOCAL MEMORY10
   SPARE_LOCAL11 : DINT ;	//SPRE LOCAL MEMORY11
   SPARE_LOCAL12 : DINT ;	//SPRE LOCAL MEMORY12
   SPARE_LOCAL13 : DINT ;	//SPRE LOCAL MEMORY13
   SPARE_LOCAL14 : INT ;	//SPRE LOCAL MEMORY14
   SPARE_LOCAL15 : INT ;	//SPRE LOCAL MEMORY15
   COMPRSR_1_2_SELC_SW : BOOL ;	//COMPRESSOR 1 & 2 SELECTION
   COMPRSR_1_START_PB : BOOL ;	//COMPRESSOR 1 START PUSH BUTTON
   COMPRSR_1_RDY_START : BOOL ;	//COMPRESSOR 1 READY TO START
   COMPRSR_1_STOP_PB : BOOL ;	//COMPRESSOR 1 STOP PUSH BUTTON
   COMPRSR_CNTRL_PS2_SW_FB : BOOL ;	//COMPRESSOR CONTROL PRESSURE SWITCH2 FEED BACK
   COMPRSR_2_START_PB : BOOL ;	//COMPRESSOR 2 START PUSH BUTTON
   COMPRSR_2_RDY_START : BOOL ;	//COMPRESSOR 2 READY TO START
   COMPRSR_2_STOP_PB : BOOL ;	//COMPRESSOR 2 STOP PUSH BUTTON
   COMPRSR_EMER_PRESSED : BOOL ;	//COMPRESSOR EMERGENCY PRESSED BIT
   COMPRSR_1_RUNNG_FB : BOOL ;	//COMPRESSOR 1 RUNNING FEED BACK
   COMPRSR_2_RUNNG_FB : BOOL ;	//COMPRESSOR 2 RUNNING FEED BACK
   ALARM_ACT_PB_AT_CD : BOOL ;	//ALARM ACKNOWLODGE PUSH BUTTON AT CD
   LAMP_TECT_PB_AT_CD : BOOL ;	//LAMP TEST PUSH BUTTON AT CD
   COMPRSR_MAX_PS_SW_FB : BOOL ;	//COMPRESSOR MAX PRESSURE SWITCH1 FEED BACK
   SPARE_INPUT1 : INT ;	//SPARE INPUT 1
   SPARE_INPUT2 : INT ;	//SPARE INPUT 2
   SPARE_INPUT3 : INT ;	//SPARE INPUT 3
   SPARE_INPUT4 : INT ;	//SPARE INPUT 4
   COMPRSR_1_ON_CMD : BOOL ;	//COMPRESSOR 1 ON COMMEND
   COMPRSR_2_ON_CMD : BOOL ;	//COMPRESSOR 2 ON COMMEND
   COMPRSR_1_ON_IND : BOOL ;	//COMPRESSOR 1 ON INDICATION
   COMPRSR_2_ON_IND : BOOL ;	//COMPRESSOR 2 ON INDICATION
  END_STRUCT ;	
BEGIN
END_DATA_BLOCK

DATA_BLOCK "PROFIBUS_DATA"	// DB 10
AUTHOR : VMK
FAMILY : MEGATECH
VERSION : 0.1
  STRUCT
   TRVLDRV1_RESERVED1_BIT : BOOL ;	//TRAVEL DRIVE-1 RESERVED1 BIT
   TRVLDRV1_PROFI_SELECTED : BOOL ;	//TRAVEL DRIVE-1 PROFIBUS SELECTED BIT
   TRVLDRV1_REF_REACHED_BIT : BOOL ;	//TRAVEL DRIVE-1 REFERENCE REACHED BIT
   TRVLDRV1_RESERVED2_BIT : BOOL ;	//TRAVEL DRIVE-1 RESERVED2 BIT
   TRVLDRV1_RESERVED3_BIT : BOOL ;	//TRAVEL DRIVE-1 RESERVED3 BIT
   TRVLDRV1_RESERVED4_BIT : BOOL ;	//TRAVEL DRIVE-1 RESERVED4 BIT
   TRVLDRV1_RESERVED5_BIT : BOOL ;	//TRAVEL DRIVE-1 RESERVED5 BIT
   TRVLDRV1_REVERSE_DIR_BIT : BOOL ;	//TRAVEL DRIVE-1 REVERSE DIRECTION BIT
   TRVLDRV1_RDY_SWITCH_ON : BOOL ;	//TRAVEL DRIVE-1 READY TO SWITCH ON BIT
   TRVLDRV1_RDY_BIT : BOOL ;	//TRAVEL DRIVE-1 READY BIT
   TRVLDRV1_RUNNING_BIT : BOOL ;	//TRAVEL DRIVE-1 RUNNING BIT
   TRVLDRV1_FAULT_BIT : BOOL ;	//TRAVEL DRIVE-1 FAULT BIT
   TRVLDRV1_VOLTAGE_ENABLE : BOOL ;	//TRAVEL DRIVE-1 VOLTAGE ENABLED BIT
   TRVLDRV1_EMGSTOP_BIT : BOOL ;	//TRAVEL DRIVE-1 EMERGENCY STOP BIT
   TRVLDRV1_SWTCHON_DISABLE : BOOL ;	//TRAVEL DRIVE-1 SWITCH ON DISABLE BIT
   TRVLDRV1_ALARM_BIT : BOOL ;	//TRAVEL DRIVE-1 ALARM BIT
   TRVLDRV1_SPEED_ACTUAL : INT ;	//TRAVEL DRIVE-1 SPEED ACTUAL VALUE
   TRVLDRV1_CONTROLWORD : WORD ;	//TRAVEL DRIVE-1 CONTROL WORD VALUE
   TRVLDRV1_SPEED_REF : INT ;	//TRVVEL DRIVE-1 SPEED REFERENCE VALUE
   TRVLDRV2_RESERVED1_BIT : BOOL ;	//TRAVEL DRIVE-2 RESERVED1 BIT
   TRVLDRV2_PROFI_SELECTED : BOOL ;	//TRAVEL DRIVE-2 PROFIBUS SELECTED BIT
   TRVLDRV2_REF_REACHED_BIT : BOOL ;	//TRAVEL DRIVE-2 REFERENCE REACHED BIT
   TRVLDRV2_RESERVED2_BIT : BOOL ;	//TRAVEL DRIVE-2 RESERVED2 BIT
   TRVLDRV2_RESERVED3_BIT : BOOL ;	//TRAVEL DRIVE-2 RESERVED3 BIT
   TRVLDRV2_RESERVED4_BIT : BOOL ;	//TRAVEL DRIVE-2 RESERVED4 BIT
   TRVLDRV2_RESERVED5_BIT : BOOL ;	//TRAVEL DRIVE-2 RESERVED5 BIT
   TRVLDRV2_REVERSE_DIR_BIT : BOOL ;	//TRAVEL DRIVE-1 REVERSE DIRECTION BIT
   TRVLDRV2_RDY_SWITCH_ON : BOOL ;	//TRAVEL DRIVE-2 READY TO SWITCH ON BIT
   TRVLDRV2_RDY_BIT : BOOL ;	//TRAVEL DRIVE-2 READY BIT
   TRVLDRV2_RUNNING_BIT : BOOL ;	//TRAVEL DRIVE-2 RUNNING BIT
   TRVLDRV2_FAULT_BIT : BOOL ;	//TRAVEL DRIVE-2 FAULT BIT
   TRVLDRV2_VOLTAGE_ENABLE : BOOL ;	//TRAVEL DRIVE-2 VOLTAGE ENABLED BIT
   TRVLDRV2_EMGSTOP_BIT : BOOL ;	//TRAVEL DRIVE-2 EMERGENCY STOP BIT
   TRVLDRV2_SWTCHON_DISABLE : BOOL ;	//TRAVEL DRIVE-2 SWITCH ON DISABLE BIT
   TRVLDRV2_ALARM_BIT : BOOL ;	//TRAVEL DRIVE-2 ALARM BIT
   TRVLDRV2_SPEED_ACTUAL : INT ;	//TRAVEL DRIVE-2 SPEED ACTUAL VALUE
   TRVLDRV2_CONTROLWORD : WORD ;	//TRAVEL DRIVE-2 CONTROL WORD VALUE
   TRVLDRV2_SPEED_REF : INT ;	//TRVVEL DRIVE-2 SPEED REFERENCE VALUE
  END_STRUCT ;	
BEGIN
   TRVLDRV2_CONTROLWORD := W#16#477;
END_DATA_BLOCK

DATA_BLOCK "CMD_FROM_TATA"	// DB 11
VERSION : 0.1
  STRUCT
   QL_OnBord_STATUS_BIT : STRUCT
    PC_ILK_OK : BOOL ;	//Pushing interlock OK
    QL_LT_MODE : BOOL ;	//Long travel in auto or in man
    QL_TRAVEL_FWD : BOOL ;	//FWD over profibus
    QL_TRAVEL_REV : BOOL ;	//REV over profibus
    QL_TRAVEL_START : BOOL ;	//START over profibus
    QL_TRAVEL_STOP : BOOL ;	//STOP  over profibus
    QL_CripeSpeed : BOOL ;
    QL_LIGHT_ON_CMD : BOOL ;	//LIGHT ON COMMAND
    SpareBit_3 : BOOL ;
    SpareBit_4 : BOOL ;
    SpareBit_5 : BOOL ;
    SpareBit_6 : BOOL ;
    SpareBit_7 : BOOL ;
    SpareBit_8 : BOOL ;
    SpareBit_9 : BOOL ;
    SpareBit_10 : BOOL ;
    PC_SPEED_REF : INT ;	//Reserve for LT motion (spd_ref) over profibus
    SATA : ARRAY  [1 .. 7 ] OF INT ;
   END_STRUCT ;
  END_STRUCT ;	
BEGIN
END_DATA_BLOCK

DATA_BLOCK "FB_TO_TATA"	// DB 12
VERSION : 0.1
  STRUCT
   QL_MACHINE_STATUS_BIT : STRUCT
    QL_Permissive : BOOL ;	//QL READY FOR TRAVEL
    QL_COB1 : BOOL ;
    QL_COB2 : BOOL ;
    QL_DRV_STATU : BOOL ;	//Drive healthy/unhealthy
    QL_DRV_FWD : BOOL ;	//Motion towards quenching tower
    QL_DRV_REV : BOOL ;	//Motion towards coal tower
    QL_READY : BOOL ;	//QUINCHING LOCO READY
    TRAVEL_MODE : BOOL ;	//TRAVEL MODE SELECTED IN AUTO
    Spare2 : BOOL ;
    Spare3 : BOOL ;
    Spare4 : BOOL ;
    Spare5 : BOOL ;
    Spare7 : BOOL ;
    Spare8 : BOOL ;
    Spare9 : BOOL ;
    Spare10 : BOOL ;
    SpareInt0 : INT ;
    QL_PUSH_SPEED : REAL ;	//QUENCHING LOCO SPEED FEEDBACK
    SpareInt1 : INT ;
    SATA : ARRAY  [1 .. 4 ] OF INT ;
   END_STRUCT ;
  END_STRUCT ;	
BEGIN
END_DATA_BLOCK

DATA_BLOCK "FLAPPER_GATE_DB"	// DB 13
VERSION : 0.1
  STRUCT
   FLAP_GATE_1_CLS_FB : BOOL ;	//FLAPPER GATE 1 CLOSE FEED BACK
   FLAP_GATE_2_CLS_FB : BOOL ;	//FLAPPER GATE 2 CLOSE FEED BACK
   FLAP_GATE_1_CLS_IND : BOOL ;	//FLAPPER GATE 1 CLOSE INDICATION
   FLAP_GATE_2_CLS_IND : BOOL ;	//FLAPPER GATE 2 CLOSE INDICATION
   FLAP_GATE_1_OPN_IND : BOOL ;	//FLAPPER GATE 1 OPEN INDICATION
   FLAP_GATE_2_OPN_IND : BOOL ;	//FLAPPER GATE 2 OPEN INDICATION
   QL_NOT_RDY_INPUT : BOOL ;	//QUENCHING LOCO NOT READY INPUT
  END_STRUCT ;	
BEGIN
END_DATA_BLOCK

DATA_BLOCK "RECEIVE_DB_342-5"	// DB 21
VERSION : 0.1
BEGIN
// 12 bytes; values not shown
END_DATA_BLOCK

DATA_BLOCK "SEND_DB_342-5"	// DB 22
VERSION : 0.1
BEGIN
// 18 bytes; values not shown
END_DATA_BLOCK

DATA_BLOCK "SPARE_1_DB"	// DB 89
VERSION : 0.1
  STRUCT
   SPARE1 : DINT ;
   SPARE2 : DINT ;
   SPARE3 : DINT ;
   SPARE4 : DINT ;
   SPARE5 : DINT ;
   SPARE6 : DINT ;
   SPARE7 : DINT ;
   SPARE8 : DINT ;
   SPARE9 : DINT ;
   SPARE10 : DINT ;
   SPARE11 : DINT ;
   SPARE12 : DINT ;
   SPARE13 : DINT ;
   SPARE14 : DINT ;
   SPARE15 : DINT ;
   SPARE16 : DINT ;
   SPARE17 : DINT ;
   SPARE18 : DINT ;
   SPARE19 : INT ;
   SPARE20 : BOOL ;
   SPARE20_1 : BOOL ;
   SPARE21 : DINT ;
   SPARE22 : DINT ;
   SPARE23 : DINT ;
   SPARE24 : DINT ;
   SPARE25 : INT ;
   SPARE26 : DINT ;
   SPARE27 : DINT ;
   SPARE28 : DINT ;
   SPARE29 : DINT ;
   SPARE30 : DINT ;
   SPARE31 : DINT ;
   SPARE32 : DINT ;
   SPARE33 : BOOL ;
   SPARE33_1 : BOOL ;
   SPARE33_2 : BOOL ;
   SPARE33_3 : BOOL ;
   SPARE33_4 : BOOL ;
   SPARE33_5 : BOOL ;
   SPARE33_6 : BOOL ;
   SPARE33_7 : BOOL ;
   SPARE34 : DINT ;
   SPARE35 : DINT ;
   SPARE36 : DINT ;
   SPARE37 : DINT ;
   SPARE38 : INT ;
   SPARE39 : INT ;
   SPARE40 : DINT ;
   SPARE41 : DINT ;
   SPARE42 : DINT ;
   SPARE43 : DINT ;
   SPARE44 : DINT ;
   SPARE45 : DINT ;
   SPARE46 : DINT ;
   SPARE47 : BOOL ;
   SPARE47_1 : BOOL ;
   SPARE48 : INT ;
   SPARE489 : INT ;
  END_STRUCT ;	
BEGIN
END_DATA_BLOCK

DATA_BLOCK "SPARE_2_DB"	// DB 90
VERSION : 0.1
  STRUCT
   SPARE1 : INT ;
   SPARE2 : INT ;
   SPARE3 : DINT ;
   SPARE4 : DINT ;
   SPARE5 : DINT ;
   SPARE6 : DINT ;
   SPARE7 : DINT ;
   SPARE8 : DINT ;
   SPARE9 : DINT ;
   SPARE10 : DINT ;
   SPARE11 : DINT ;
   SPARE12 : DINT ;
   SPARE13 : DINT ;
   SPARE14 : DINT ;
   SPARE15 : DINT ;
   SPARE16 : DINT ;
   SPARE17 : DINT ;
   SPARE18 : DINT ;
   SPARE19 : DINT ;
   SPARE20 : DINT ;
   SPARE21 : DINT ;
  END_STRUCT ;	
BEGIN
END_DATA_BLOCK

ORGANIZATION_BLOCK "CYCLIC_EXECUCTION"	// OB 1
VERSION : 0.1
BEGIN
// (block stored without names or comments; labels and parameter names are numbered)
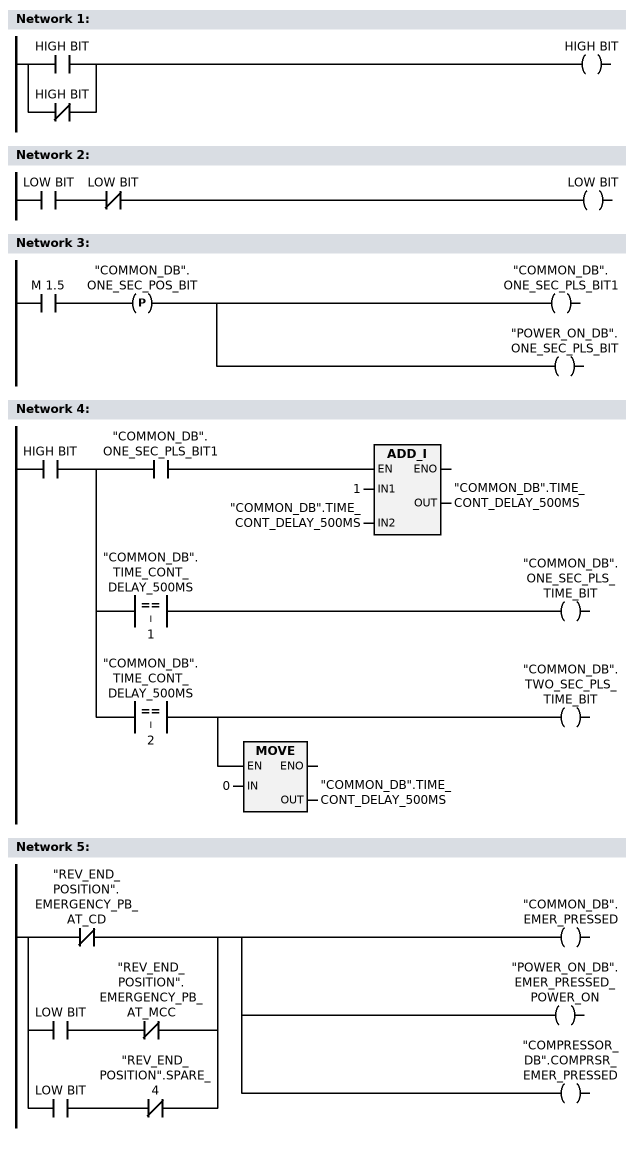
NETWORK
TITLE =
      O     "HIGH BIT";
      ON    "HIGH BIT";
      =     "HIGH BIT";
NETWORK
TITLE =
      A     "LOW BIT";
      AN    "LOW BIT";
      =     "LOW BIT";
NETWORK
TITLE =
      A     M 1.5;
      FP    "COMMON_DB".ONE_SEC_POS_BIT;
      =     "COMMON_DB".ONE_SEC_PLS_BIT1;
      =     "POWER_ON_DB".ONE_SEC_PLS_BIT;
NETWORK
TITLE =
      A     "HIGH BIT";
      =     L 20.0;
      A     L 20.0;
      A     "COMMON_DB".ONE_SEC_PLS_BIT1;
      JNB   M001;
      L     1;
      L     "COMMON_DB".TIME_CONT_DELAY_500MS;
      +I;
      T     "COMMON_DB".TIME_CONT_DELAY_500MS;
M001: NOP   0;
      A     L 20.0;
      A(;
      L     "COMMON_DB".TIME_CONT_DELAY_500MS;
      L     1;
      ==I;
      );
      =     "COMMON_DB".ONE_SEC_PLS_TIME_BIT;
      A     L 20.0;
      A(;
      L     "COMMON_DB".TIME_CONT_DELAY_500MS;
      L     2;
      ==I;
      );
      =     L 20.1;
      A     L 20.1;
      BLD   102;
      =     "COMMON_DB".TWO_SEC_PLS_TIME_BIT;
      A     L 20.1;
      JNB   M002;
      L     0;
      T     "COMMON_DB".TIME_CONT_DELAY_500MS;
M002: NOP   0;
NETWORK
TITLE =
      ON    "REV_END_POSITION".EMERGENCY_PB_AT_CD;
      O;
      A     "LOW BIT";
      AN    "REV_END_POSITION".EMERGENCY_PB_AT_MCC;
      O;
      A     "LOW BIT";
      AN    "REV_END_POSITION".SPARE_4;
      =     "COMMON_DB".EMER_PRESSED;
      =     "POWER_ON_DB".EMER_PRESSED_POWER_ON;
      =     "COMPRESSOR_DB".COMPRSR_EMER_PRESSED;
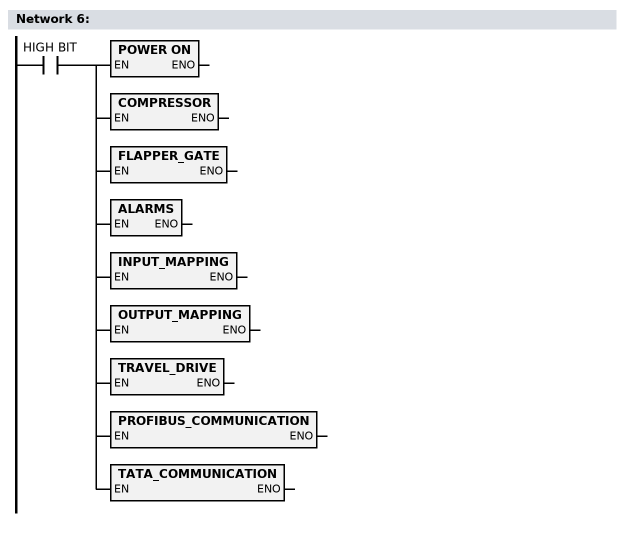
NETWORK
TITLE =
      A     "HIGH BIT";
      =     L 20.0;
      A     L 20.0;
      JNB   M003;
      CALL  "POWER ON";
M003: NOP   0;
      A     L 20.0;
      JNB   M004;
      CALL  "COMPRESSOR";
M004: NOP   0;
      A     L 20.0;
      JNB   M005;
      CALL  "FLAPPER_GATE";
M005: NOP   0;
      A     L 20.0;
      JNB   M006;
      CALL  "ALARMS";
M006: NOP   0;
      A     L 20.0;
      JNB   M007;
      CALL  "INPUT_MAPPING";
M007: NOP   0;
      A     L 20.0;
      JNB   M008;
      CALL  "OUTPUT_MAPPING";
M008: NOP   0;
      A     L 20.0;
      JNB   M009;
      CALL  "TRAVEL_DRIVE";
M009: NOP   0;
      A     L 20.0;
      JNB   M010;
      CALL  "PROFIBUS_COMMUNICATION";
M010: NOP   0;
      A     L 20.0;
      JNB   M011;
      CALL  "TATA_COMMUNICATION";
M011: NOP   0;
END_ORGANIZATION_BLOCK

ORGANIZATION_BLOCK "CYCL_FLT"	// OB 80
VERSION : 0.1
BEGIN
// (block stored without names or comments; labels and parameter names are numbered)
NETWORK
TITLE =
      NOP   0;
END_ORGANIZATION_BLOCK

ORGANIZATION_BLOCK "I/O_FLT1"	// OB 82
VERSION : 0.1
BEGIN
// (block stored without names or comments; labels and parameter names are numbered)
NETWORK
TITLE =
      NOP   0;
END_ORGANIZATION_BLOCK

ORGANIZATION_BLOCK "OBNL_FLT"	// OB 85
VERSION : 0.1
BEGIN
// (block stored without names or comments; labels and parameter names are numbered)
NETWORK
TITLE =
      NOP   0;
END_ORGANIZATION_BLOCK

ORGANIZATION_BLOCK "RACK_FLT"	// OB 86
VERSION : 0.1
BEGIN
// (block stored without names or comments; labels and parameter names are numbered)
END_ORGANIZATION_BLOCK

ORGANIZATION_BLOCK "COMM_FLT"	// OB 87
VERSION : 0.1
BEGIN
// (block stored without names or comments; labels and parameter names are numbered)
NETWORK
TITLE =
      NOP   0;
END_ORGANIZATION_BLOCK

ORGANIZATION_BLOCK "COMPLETE RESTART"	// OB 100
VERSION : 0.1
BEGIN
// (block stored without names or comments; labels and parameter names are numbered)
END_ORGANIZATION_BLOCK

ORGANIZATION_BLOCK "PROG_ERR"	// OB 121
VERSION : 0.1
BEGIN
// (block stored without names or comments; labels and parameter names are numbered)
END_ORGANIZATION_BLOCK

ORGANIZATION_BLOCK "MOD_ERR"	// OB 122
VERSION : 0.1
BEGIN
// (block stored without names or comments; labels and parameter names are numbered)
NETWORK
TITLE =
      NOP   0;
END_ORGANIZATION_BLOCK
